// TwinCAT 3 PLC project TcoCoreTests
// Title: TcoCoreTests
// Company: Vortex.Library
// ProjectVersion: 0.6.0.913
// ProgramVersion: 3.1.4024.12
// libraries:
//   Tc2_EtherCAT, * (Beckhoff Automation GmbH)
//   Tc2_Standard, * (Beckhoff Automation GmbH)
//   Tc2_System, * (Beckhoff Automation GmbH)
//   Tc3_Module, * (Beckhoff Automation GmbH)
//   TcoCore, 0.6.0.913 (Vortex.Library)
// project tree:
//   Components/ fbPiston.TcPOU, fbPistonConfig.TcDUT, fbPistonMoveTask.TcPOU, fbPistonStatus.TcDUT, IPistonGripper.TcIO, IPistonHorizontal.TcIO, IPistonVertical.TcIO
//   / PlcTask1.TcTTO
//   POUs/ MAIN.TcPOU
//   Tests/TcoComponent/PlcExecuted/ eTcoComponentTests.TcDUT, TcoComponentTestContext.TcPOU, TestComponent.TcPOU
//   Tests/TcoComponent/ TcoComponentTest.TcPOU, _TcoComponent.TcPOU
//   Tests/TcoContext/ TcoContextTest.TcPOU
//   Tests/TcoLogger/PlcExecuted/ eTcoLoggerTests.TcDUT, TcoLoggerTestContext.TcPOU, TcoLoggerTest.TcPOU
//   Tests/TcoMessenger/ TcoContextMessagingPerf.TcPOU, TcoMessengerContextTest.TcPOU, TcoMessengerTests.TcPOU
//   Tests/TcoObject/EqualsOverride/ TcoObjectEqualsTest.TcPOU
//   Tests/TcoObject/ TcoObjectTest.TcPOU
//   Tests/TcoRemoteTask/PlcExecuted/ eTcoRemoteTaskTests.TcDUT, TcoRemoteTaskTest.TcPOU, TcoRemoteTaskTestContext.TcPOU
//   Tests/TcoRtc/ TcoRtcTest.TcPOU
//   Tests/TcoSequenceObserver/ eTcoSequenceObserverTests.TcDUT, TcoSequenceObserverTests.TcPOU
//   Tests/TcoSequencer/PlcExecuted/ eTcoSequencerTests.TcDUT, TcoSequencerTestChildState.TcPOU, TcoSequencerTestContext.TcPOU, TcoSequencerTestType.TcPOU
//   Tests/TcoSequencer/ TcoSequencerAutoRestorableTest.TcPOU, TcoSequencerNonAutoRestorableTest.TcPOU, _TcoSequencer.TcPOU
//   Tests/TcoSequence/PlcExecuted/ eTcoSequenceTests.TcDUT, TcoSequenceTestChildState.TcPOU, TcoSequenceTestContext.TcPOU, TcoSequenceTestType.TcPOU
//   Tests/TcoSequence/ TcoSequenceAutoRestorableTest.TcPOU, TcoSequenceNonAutoRestorableTest.TcPOU, _TcoSequence.TcPOU
//   Tests/TcoState/ TcoStateTest.TcPOU, TcoStateAutoRestoreTest.TcPOU
//   Tests/TcoTask/PlcExecuted/ eTcoTaskTests.TcDUT, TcoTaskPlcTestState.TcPOU, TcoTaskPlcTestObject.TcPOU, TcoTaskPlcTest.TcPOU, TcoTaskTestContext.TcPOU
//   Tests/TcoTask/ TcoTaskTest.TcPOU
//   Tests/TcoToggleTask/ eTcoToggleTaskTests.TcDUT, TcoToggleTaskTestContext.TcPOU, TcoToggleTaskTests.TcPOU
//   Tests/Utilities/ StringBuilderTests.TcPOU
// (motion and I/O tree: see PLC project tcocore)
// real-time tasks:
//   TASK PlcTask: cycle T#10ms, priority 20, ADS port 350
//   TASK PlcTask1: cycle T#10ms, priority 21, ADS port 351
//   TASK PlcTask2: cycle T#10ms, priority 22, ADS port 352

CONFIGURATION TcoCoreTests
    RESOURCE PLC ON TwinCAT3
        TASK PlcTask1(INTERVAL := T#10ms, PRIORITY := 21);
        PROGRAM MAIN WITH PlcTask1 : MAIN;
    END_RESOURCE
END_CONFIGURATION

// ---- Components/fbPistonConfig.TcDUT
TYPE fbPistonConfig :
STRUCT
    MaxTimeToReachHome : TIME;
    MaxTimeToReachWork : TIME;
END_STRUCT
END_TYPE

// ---- Components/fbPistonStatus.TcDUT
TYPE fbPistonStatus :
STRUCT
    AtHome : TIME;
    AtWork : TIME;
END_STRUCT
END_TYPE

// ---- Tests/TcoComponent/PlcExecuted/eTcoComponentTests.TcDUT
{attribute 'qualified_only'}
{attribute 'strict'}
TYPE eTcoComponentTests :
(
    GetSignalInfo := 100
);
END_TYPE

// ---- Tests/TcoLogger/PlcExecuted/eTcoLoggerTests.TcDUT
{attribute 'qualified_only'}
{attribute 'strict'}
TYPE eTcoLoggerTests :
(
    PushMessage := 10,
    PushMessageMultiple := 20,
    PushMessageMultipleInMoreCycles := 30,
    SimplePush := 40
);
END_TYPE

// ---- Tests/TcoRemoteTask/PlcExecuted/eTcoRemoteTaskTests.TcDUT
{attribute 'qualified_only'}
{attribute 'strict'}
TYPE eTcoRemoteTaskTests :
(
    RestoreTasks := 10,
    InvokeInitializedCSharpMethod := 100,
    InvokeNotInitializedCSharpMethod := 200,
    ExceptionInMethodWillResultInException := 400
);
END_TYPE

// ---- Tests/TcoSequenceObserver/eTcoSequenceObserverTests.TcDUT
{attribute 'qualified_only'}
{attribute 'strict'}
TYPE eTcoSequenceObserverTests :
(
    RestoreSequencer := 1,
    RunSequenceWithObserverTest := 10,
    RunSequenceWithoutObserverTest := 20
);
END_TYPE

// ---- Tests/TcoSequencer/PlcExecuted/eTcoSequencerTests.TcDUT
{attribute 'qualified_only'}
{attribute 'strict'}
TYPE eTcoSequencerTests :
(
    none := -1,
    CallSequencerBodiesOnly := 100,
    RestoreSequencers,
    NumberOfStepsCount := 500,
    ExecutionInOnePLCcycle := 501,
    OnStepCompleted := 502,
    OnSequenceCompleted := 503,
    RestoreChildBetweenSteps := 504,
    OnStateChangeWithRestoreCallInside := 505,
    MinStepId := 506,
    MaxStepId := 507,
    RequestStepToFirstStepWithStepId0 := 508,
    RequestStep := 509,
    CheckStepIdUniqueness := 510,
    RestoreAlreadyCheckedSequence := 512,
    NotUniqueStepId := 513,
    AfterErrorRestore := 516,
    ChangeStepIdDuringExecution := 520,
    CommentOutPartOfRunningSequencer := 524,
    UncommentPartOfRunningSequencer := 526,
    OpenCloseSequence := 530,
    RequestStepFromLowerToHigher := 541,
    RequestStepFromHigherToLower := 542,
    RequestStepToNotExistingStep := 544,
    RequestStepWhilePreviousRequestStepHasNotBeenYetProcessed := 547,
    DisableStepEnabledAndActiveInPreviousPLCcycle := 551,
    RequestStepCallingCyclically := 560,
    SetStepMode := 570,
    StepMode := 580,
    InvalidMode := 582,
    StepInError := 583,
    CheckStepIdUniquenessStepMode := 590,
    NotUniqueStepIdInStepMode := 594,
    AfterErrorResetInStepMode := 597,
    InvalidModeDetailed := 602,
    StepInErrorDetailed := 604,
    StepModeStepIn := 611,
    StepModeChangeStepIdDuringExecution := 612,
    StepModeChangeStepOrder := 615,
    StepModeCommentOutPartOfRunningSequencer := 618,
    StepModeUncommentPartOfRunningSequencer := 621,
    StepModeRequestStepFromLowerToHigher := 631,
    StepModeRequestStepFromHigherToLower := 633,
    StepModeRequestStepToNotExistingStep := 635,
    StepModeRequestStepWhilePreviousRequestStepHasnotBeenYetProcessed := 640,
    StepModeDisabledStep := 641,
    StepModeStepForwardBackward := 670,
    StepModeStepInDetailed := 681,
    SwitchStepModeOnDuringStepExecution := 691,
    StepModeStepForwardFromRunningStep := 693,
    StepModeStepBackwardFromRunningStep := 695,
    SwitchStepModeStepOffFromReadyToRun := 696,
    SwitchStepModeStepOnFromRunning := 697,
    SwitchStepModeStepOffFromRunning := 698,
    OnStateChangeWhenChangingModes := 699
);
END_TYPE

// ---- Tests/TcoSequence/PlcExecuted/eTcoSequenceTests.TcDUT
{attribute 'qualified_only'}
{attribute 'strict'}
TYPE eTcoSequenceTests :
(
    none := -1,
    Initialize := 10,
    CallSequencerBodiesOnly := 100,
    RestoreSequencers,
    NumberOfStepsCount := 500,
    ExecutionInOnePLCcycle := 501,
    OnStepCompleted := 502,
    OnSequenceCompleted := 503,
    RestoreChildBetweenSteps := 504,
    OnStateChangeWithRestoreCallInside := 505,
    MinStepId := 506,
    MaxStepId := 507,
    RequestStepToFirstStepWithStepId0 := 508,
    RequestStep := 509,
    CheckStepIdUniqueness := 510,
    RestoreAlreadyCheckedSequence := 512,
    NotUniqueStepId := 513,
    AfterErrorRestore := 516,
    ChangeStepIdDuringExecution := 520,
    CommentOutPartOfRunningSequencer := 524,
    UncommentPartOfRunningSequencer := 526,
    OpenCloseSequence := 530,
    RequestStepFromLowerToHigher := 541,
    RequestStepFromHigherToLower := 542,
    RequestStepToNotExistingStep := 544,
    RequestStepWhilePreviousRequestStepHasNotBeenYetProcessed := 547,
    DisableStepEnabledAndActiveInPreviousPLCcycle := 551,
    RequestStepCallingCyclically := 560,
    SetStepMode := 570,
    StepMode := 580,
    InvalidMode := 582,
    StepInError := 583,
    CheckStepIdUniquenessStepMode := 590,
    NotUniqueStepIdInStepMode := 594,
    AfterErrorResetInStepMode := 597,
    InvalidModeDetailed := 602,
    StepInErrorDetailed := 604,
    StepModeStepIn := 611,
    StepModeChangeStepIdDuringExecution := 612,
    StepModeChangeStepOrder := 615,
    StepModeCommentOutPartOfRunningSequencer := 618,
    StepModeUncommentPartOfRunningSequencer := 621,
    StepModeRequestStepFromLowerToHigher := 631,
    StepModeRequestStepFromHigherToLower := 633,
    StepModeRequestStepToNotExistingStep := 635,
    StepModeRequestStepWhilePreviousRequestStepHasnotBeenYetProcessed := 640,
    StepModeDisabledStep := 641,
    StepModeStepForwardBackward := 670,
    StepModeStepInDetailed := 681,
    SwitchStepModeOnDuringStepExecution := 691,
    StepModeStepForwardFromRunningStep := 693,
    StepModeStepBackwardFromRunningStep := 695,
    SwitchStepModeStepOffFromReadyToRun := 696,
    SwitchStepModeStepOnFromRunning := 697,
    SwitchStepModeStepOffFromRunning := 698,
    OnStateChangeWhenChangingModes := 699,
    MissedSequenceOpening := 6100,
    MissedSequenceClosing := 6200,
    FreshStateEntry := 6300
);
END_TYPE

// ---- Tests/TcoTask/PlcExecuted/eTcoTaskTests.TcDUT
{attribute 'qualified_only'}
{attribute 'strict'}
TYPE eTcoTaskTests :
(
    CallTasksBodiesOnly := 100,
    RestoreTasks,
    TaskInvokeAndWaitForDone := 300,
    TaskInvokeAfterDoneWithNoEmptyCycles,
    TaskInvokeAfterDoneWithOneEmptyCycle,
    TaskInvokeAfterDoneWithAbortCall,
    TaskInvokeAfterDoneWithRestoreCall,
    TaskAbortDuringExecutionAndInvoke,
    TaskError := 310,
    TaskInvokeAfterErrorNoRestoreNoEmptyCycles,
    TaskInvokeAfterErrorNoRestoreOneEmptyCycle,
    TaskInvokeAfterErrorWithRestore,
    TaskAbortDuringExecution,
    TaskMessage,
    IdentitiesTest,
    CheckAutoRestoreProperties,
    AutoRestoreOnStateChange,
    InvokeDisabledTask := 320,
    DisableExecutingTask,
    InvokeTaskThenDisable,
    DisableTaskInErrorStateEnableAndTriggerAgain,
    ElapsedTypeMeasurement := 330,
    TaskExecutingWithDoneAndErrorStatement := 340,
    TaskExecutingWithErrorAndDoneStatement := 350,
    TaskExecuteMethodNotCalled := 360,
    TaskExecuteMethodCalled := 370
);
END_TYPE

// ---- Tests/TcoToggleTask/eTcoToggleTaskTests.TcDUT
{attribute 'qualified_only'}
{attribute 'strict'}
TYPE eTcoToggleTaskTests :
(
    Reinit := 1001,
    CleanUp := 1002,
    Message := 1003,
    TriggerToggleWhileRunNotCalled := 1004,
    TriggerToggleWhileDisabled := 1005,
    TriggerToggleWhileEnabled := 1006,
    TriggerOnWhileRunNotCalled := 1007,
    TriggerOnWhileDisabled := 1008,
    TriggerOnWhileEnabled := 1009,
    TriggerOffWhileRunNotCalled := 1010,
    TriggerOffWhileDisabled := 1011,
    TriggerOffWhileEnabled := 1012
);
END_TYPE

// ---- Components/IPistonGripper.TcIO
INTERFACE IPistonGripper

METHOD Close : TcoCore.ITcoTaskStatus
END_METHOD

METHOD Open : TcoCore.ITcoTaskStatus
END_METHOD

END_INTERFACE

// ---- Components/IPistonHorizontal.TcIO
INTERFACE IPistonHorizontal

METHOD MoveLeft : TcoCore.ITcoTaskStatus
END_METHOD

METHOD MoveRight : TcoCore.ITcoTaskStatus
END_METHOD

END_INTERFACE

// ---- Components/IPistonVertical.TcIO
INTERFACE IPistonVertical

METHOD MoveDown : TcoCore.ITcoTaskStatus
END_METHOD

METHOD MoveUp : TcoCore.ITcoTaskStatus
END_METHOD

END_INTERFACE

// ---- POUs/MAIN.TcPOU
PROGRAM MAIN
VAR
    //TcRpc tests
    _tcoRtcTest_A : TcoRtcTest;
    _tcoRtcTest_B : TcoRtcTest;
    _tcoContextTest_A : TcoContextTest;
    _tcoContextTest_B : TcoContextTest;
    _tcoSequencerAutoRestorableTest : TcoSequencerAutoRestorableTest;
    _tcoSequencerNonAutoRestorableTest : TcoSequencerNonAutoRestorableTest;
    _tcoSequenceAutoRestorableTest : TcoSequenceAutoRestorableTest;
    _tcoSequenceNonAutoRestorableTest : TcoSequenceNonAutoRestorableTest;
    _tcoMessengerContextTest : TcoMessengerContextTest;
    _tcoContextMessagingPerf : TcoContextMessagingPerf;
    _tcoComponentTest : TcoComponentTest;
    _stringBuilderTest : StringBuilderTests;
    //PLC executed tests
    _tcoTaskTestContext : TcoTaskTestContext;
    _tcoToggleTaskTestContext : TcoToggleTaskTestContext;
    {attribute addProperty Name "Test base component class"}
    _tcoComponentTestContext : TcoComponentTestContext;
    _tcoRemoteTaskTestContext : TcoRemoteTaskTestContext;
    _tcoSequencerTestContext : TcoSequencerTestContext;
    _tcoSequenceTestContext : TcoSequenceTestContext;
    _tcoLoggerTestContext : TcoLoggerTestContext;
    _tcoSequenceObserverTests : TcoSequenceObserverTests;
END_VAR

//TcRpc tests
_tcoRtcTest_A();
_tcoRtcTest_B();
_tcoContextTest_A();
_tcoContextTest_B();
_tcoSequencerAutoRestorableTest();
_tcoSequencerNonAutoRestorableTest();
_tcoSequenceAutoRestorableTest();
_tcoSequenceNonAutoRestorableTest();
_tcoMessengerContextTest();
_tcoContextMessagingPerf();
_tcoComponentTest();
_stringBuilderTest();
//PLC executed tests
_tcoTaskTestContext.ProbeRun();
_tcoToggleTaskTestContext.ProbeRun();
_tcoComponentTestContext.ProbeRun();
_tcoRemoteTaskTestContext.ProbeRun();
_tcoSequencerTestContext.ProbeRun();
_tcoSequenceTestContext.ProbeRun();
_tcoLoggerTestContext.ProbeRun();
_tcoSequenceObserverTests.ProbeRun();

END_PROGRAM

// ---- Tests/TcoRtc/TcoRtcTest.TcPOU
FUNCTION_BLOCK TcoRtcTest EXTENDS TcoCore._internals_TcoContext
VAR
    _callMyPlcInstanceSync : BOOL := FALSE;
    _callMyPlcInstanceRun : BOOL := FALSE;
    _myIdentity : ULINT;
    _nowLocal : DATE_AND_TIME;
    _nowUtc : DATE_AND_TIME;
    _rtcIsValid : BOOL := FALSE;
    _rtcIsSynchronized : BOOL := FALSE;
    _rtcSynchParamsSet : TcoCore.RtcSynchParams;
    _rtcSynchParamsGet : TcoCore.RtcSynchParams;
END_VAR

IF THIS^._callMyPlcInstanceSync THEN
    THIS^.RtcSynchronize(_rtcSynchParamsSet.doSynch, _rtcSynchParamsSet.syncAmsId, _rtcSynchParamsSet.syncPeriod);
END_IF

IF THIS^._callMyPlcInstanceRun THEN
    THIS^.Run();
    _nowLocal := THIS^.RealTimeClock.NowLocal();
    _nowUtc := THIS^.RealTimeClock.NowUTC();
    _rtcIsValid := THIS^.RealTimeClock.IsValid;
    _rtcIsSynchronized := THIS^.RealTimeClock.IsSynchronized;
    _myIdentity := THIS^.Identity;
END_IF

{attribute 'TcRpcEnable'}
METHOD INTERNAL GetSynchParams
_rtcSynchParamsGet := SUPER^._GetSynchParams();
END_METHOD

METHOD PROTECTED Main
END_METHOD

{attribute 'TcRpcEnable'}
METHOD INTERNAL NowLocal
_nowLocal := THIS^.RealTimeClock.NowLocal();
END_METHOD

{attribute 'TcRpcEnable'}
METHOD INTERNAL NowUtc
_nowUtc := THIS^.RealTimeClock.NowUTC();
END_METHOD

{attribute 'TcRpcEnable'}
METHOD INTERNAL RtcIsSynchronized : BOOL
RtcIsSynchronized := THIS^.RealTimeClock.IsSynchronized;
_rtcIsSynchronized := THIS^.RealTimeClock.IsSynchronized;
END_METHOD

{attribute 'TcRpcEnable'}
METHOD INTERNAL RtcIsValid : BOOL
RtcIsValid := THIS^.RealTimeClock.IsValid;
_rtcIsValid := THIS^.RealTimeClock.IsValid;
END_METHOD

{attribute 'TcRpcEnable'}
METHOD INTERNAL TickClock : STRING
TickClock := Tc2_EtherCAT.DCTIME64_TO_STRING(THIS^.RealTimeClock.TickClock());
END_METHOD

END_FUNCTION_BLOCK

// ---- Tests/TcoContext/TcoContextTest.TcPOU
FUNCTION_BLOCK TcoContextTest EXTENDS TcoCore._internals_TcoContext
VAR
    _callMyPlcInstance : BOOL := FALSE;
    _startCycles : ULINT;
    _endCycles : ULINT;
    _mainCycles : ULINT;
    _tcoObjectTest_A : TcoObjectTest(THIS^);
    _tcoObjectTest_B : TcoObjectTest(THIS^);
    _tcoObjectTest_Misc : TcoObjectTest(THIS^);
    _myIdentity : ULINT;
    _onEntryCount : ULINT;
    _onExitCount : ULINT;
END_VAR

IF THIS^._callMyPlcInstance THEN
    THIS^.Run();
END_IF

{attribute 'TcRpcEnable'}
METHOD INTERNAL CallMainFromUnitTest
THIS^.Main();
END_METHOD

{attribute 'TcRpcEnable'}
METHOD INTERNAL CallRunFromUnitTest
THIS^.Run();
END_METHOD

{attribute 'TcRpcEnable'}
METHOD INTERNAL ContextClose
SUPER^._Close();
END_METHOD

{attribute 'TcRpcEnable'}
METHOD INTERNAL ContextOpen
SUPER^._Open();
END_METHOD

METHOD PROTECTED Main
_mainCycles := _mainCycles + 1;
_myIdentity := THIS^.Identity;
END_METHOD

(*~
    <docu>
        <summary>
            Called on entry into context. When overridden in derived class allows to execute an arbitrary logic prior to opening the context cycle.
            <remarks>
                <note type="important">
                    The method executes prior to opening the context. The context might not be properly initialized on first call.
                    Any information contained in the context at this point are from the last execution.
                </note>
            </remarks>
        </summary>
    </docu>
~*)
METHOD PROTECTED OnEntry
_onEntryCount := _onEntryCount + 1;
END_METHOD

(*~
    <docu>
        <summary>
            Called upon exit from the context. When overridden in derived class allows to execute an arbitrary logic after closing the context cycle.
        </summary>
    </docu>
~*)
METHOD PROTECTED OnExit
_onExitCount := _onExitCount + 1;
END_METHOD

{attribute 'TcRpcEnable'}
METHOD INTERNAL ReadOutCycleCounters
_startCycles := THIS^.StartCycleCount;
_endCycles := THIS^.EndCycleCount;
_myIdentity := THIS^.Identity;
END_METHOD

END_FUNCTION_BLOCK

// ---- Tests/TcoObject/TcoObjectTest.TcPOU
FUNCTION_BLOCK TcoObjectTest EXTENDS TcoCore.TcoObject
VAR
    _myIdentity : ULINT;
    _myContextIdentity : ULINT;
    _myContextStartCount : ULINT;
    _myContextEndCount : ULINT;
    _myParentIdentity : ULINT;
    _tcoTaskTest_A : TcoTaskTest(THIS^);
    _tcoTaskTest_B : TcoTaskTest(THIS^);
    _tcoStateTest_A : TcoStateTest(THIS^, eRestoreMode.AutoRestoreMembers);
    _tcoStateTest_B : TcoStateTest(THIS^, eRestoreMode.None);
    // Object equality
    _tcoObjectEqualsTestObj1 : TcoObjectEqualsTest(THIS^);
    _tcoObjectEqualsTestObj2 : TcoObjectEqualsTest(THIS^);
END_VAR

{attribute 'TcRpcEnable'}
METHOD INTERNAL CallTaskInstancies
_tcoTaskTest_A();
_tcoTaskTest_B();
END_METHOD

{attribute 'TcRpcEnable'}
METHOD PUBLIC EqualsOverrideTest : BOOL
EqualsOverrideTest := _tcoObjectEqualsTestObj1.EqualsTo(_tcoObjectEqualsTestObj2);
END_METHOD

{attribute 'TcRpcEnable'}
METHOD PUBLIC EqualsTest : BOOL
VAR_INPUT
    _case : INT;
END_VAR
VAR
    referenceTo_a_TcoStateTest : REFERENCE TO TcoStateTest;
END_VAR
CASE _case OF
    0:
        referenceTo_a_TcoStateTest REF= _tcoStateTest_A;
        EqualsTest := _tcoStateTest_A.EqualsTo(referenceTo_a_TcoStateTest);
    1:
        EqualsTest := _tcoStateTest_A.EqualsTo(_tcoStateTest_B);
    4:
        EqualsTest := _tcoStateTest_B.EqualsTo(_tcoStateTest_A);
    2:
        EqualsTest := _tcoObjectEqualsTestObj1.EqualsTo(_tcoObjectEqualsTestObj1);
    3:
        EqualsTest := _tcoObjectEqualsTestObj1.EqualsTo(_tcoObjectEqualsTestObj2);
END_CASE
END_METHOD

{attribute 'TcRpcEnable'}
METHOD INTERNAL ReadOutIdentities
_myIdentity := THIS^.Identity;
_myContextIdentity := THIS^.Context.Identity;
_myContextStartCount := THIS^.Context.StartCycleCount;
_myContextEndCount := THIS^.Context.EndCycleCount;
_myParentIdentity := THIS^.Parent.Identity;
END_METHOD

END_FUNCTION_BLOCK

// ---- Tests/TcoTask/TcoTaskTest.TcPOU
FUNCTION_BLOCK TcoTaskTest EXTENDS TcoCore.TcoTask
VAR
    _isBusy : BOOL;
    _isError : BOOL;
    _isDone : BOOL;
    _isReady : BOOL;
    _isInvokeRequestTrue : BOOL;
    _counterSetValue : ULINT;
    _counterValue : ULINT;
    _invokeCounter : ULINT;
    _executeCounter : ULINT;
    _doneCounter : ULINT;
    _invokeRisingEdgeCounter : ULINT;
    _executeRisingEdgeCounter : ULINT;
    _doneRisingEdgeCounter : ULINT;
    _previousState : eTaskState;
    _counterValuePV : ULINT;
    _myIdentity : ULINT;
    _myContextIdentity : ULINT;
    _myContextStartCount : ULINT;
    _myContextEndCount : ULINT;
    _myParentIdentity : ULINT;
    _autoRestoreByMyParentEnabled : BOOL;
    _onErrorCounter : ULINT;
    _whileErrorCounter : ULINT;
    _onStartCounter : ULINT;
END_VAR

ExecutionBody();

{attribute 'TcRpcEnable'}
METHOD INTERNAL Disable
THIS^.Enabled := FALSE;
END_METHOD

{attribute 'TcRpcEnable'}
METHOD INTERNAL Enable
THIS^.Enabled := TRUE;
END_METHOD

{attribute 'TcRpcEnable'}
METHOD INTERNAL ExecutionBody
IF (THIS^._taskState = eTaskState.Requested) THEN
    _invokeCounter := _invokeCounter + 1;
END_IF;

IF (THIS^._taskState = eTaskState.Requested AND _PreviousState <> eTaskState.Requested) THEN
    _counterValue := _counterSetValue;
    _counterValuePV := _counterValue;
    _invokeRisingEdgeCounter := _invokeRisingEdgeCounter + 1;
END_IF

IF (THIS^._taskState = eTaskState.Busy AND _previousState <> eTaskState.Busy) THEN
    _executeRisingEdgeCounter := _executeRisingEdgeCounter + 1;
END_IF

_previousState := THIS^._taskState;

IF (Execute()) THEN
    _executeCounter := _executeCounter + 1;
    _counterValue := _counterValue - 1;
    DoneWhen(_counterValue <= 0);
    ThrowWhen(ABS(_counterValuePV - _counterValue) > 1);
    _CounterValuePV := _counterValue;
END_IF

IF (THIS^._taskState = eTaskState.Done) THEN
    _doneCounter := _doneCounter + 1;
END_IF;

IF (THIS^._taskState = eTaskState.Done AND _previousState <> eTaskState.Done) THEN
    _doneRisingEdgeCounter := _doneRisingEdgeCounter + 1;
END_IF
END_METHOD

{attribute 'TcRpcEnable'}
METHOD INTERNAL GetMessage : STRING
GetMessage := SUPER^._messenger._mime.Text;
END_METHOD

METHOD PROTECTED OnError
_onErrorCounter := _onErrorCounter + 1;
END_METHOD

METHOD PROTECTED OnStart
_onStartCounter := _onStartCounter + 1;
END_METHOD

{attribute 'TcRpcEnable'}
METHOD INTERNAL PostMessage
VAR_INPUT
    Message : STRING;
END_VAR
THIS^.Messenger.Post(Message, eMessageCategory.Error);
END_METHOD

{attribute 'TcRpcEnable'}
METHOD INTERNAL ReadOutAutoRestoreProperties
_autoRestoreByMyParentEnabled := THIS^.AutoRestorable;
END_METHOD

{attribute 'TcRpcEnable'}
METHOD INTERNAL ReadOutIdentities
_myIdentity := THIS^.Identity;
_myContextIdentity := THIS^.Context.Identity;
_myContextStartCount := THIS^.Context.StartCycleCount;
_myContextEndCount := THIS^.Context.EndCycleCount;
_myParentIdentity := THIS^.Parent.Identity;
END_METHOD

{attribute 'TcRpcEnable'}
METHOD INTERNAL ReadOutState
_isBusy := THIS^.Busy;
_isError := THIS^.Error;
_isDone := THIS^.Done;
_isReady := THIS^.Ready;
_isInvokeRequestTrue := THIS^._invokeRequest;
END_METHOD

{attribute 'TcRpcEnable'}
METHOD INTERNAL SetInvokeRequest
THIS^._invokeRequest := TRUE;
END_METHOD

{attribute 'TcRpcEnable'}
METHOD INTERNAL SetPreviousStateToReady
THIS^._previousState := eTaskState.Ready;
END_METHOD

{attribute 'TcRpcEnable'}
METHOD INTERNAL TriggerAbort
THIS^.Abort();
END_METHOD

{attribute 'TcRpcEnable'}
METHOD INTERNAL TriggerInvoke
THIS^.Invoke();
END_METHOD

{attribute 'TcRpcEnable'}
METHOD INTERNAL TriggerRestore
THIS^.Restore();
END_METHOD

(*~
    <docu>
        <summary>
            Executes until task is in ```Error``` state .
        </summary>
    </docu>
~*)
METHOD PROTECTED WhileError
_whileErrorCounter := _whileErrorCounter + 1;
END_METHOD

END_FUNCTION_BLOCK

// ---- Tests/TcoState/TcoStateTest.TcPOU
FUNCTION_BLOCK TcoStateTest EXTENDS TcoState
VAR
    _myIdentity : ULINT;
    _myContextIdentity : ULINT;
    _myContextStartCount : ULINT;
    _myContextEndCount : ULINT;
    _myParentIdentity : ULINT;
    _myState : INT;
    _tcoTaskTest_A : TcoTaskTest(THIS^);
    _tcoTaskTest_B : TcoTaskTest(THIS^);
    _tcoStateTest_A : TcoStateAutoRestoreTest(THIS^, eRestoreMode.None);
    _tcoStateTest_B : TcoStateAutoRestoreTest(THIS^, eRestoreMode.None);
    _onStateChangeCounter : INT;
    _autoRestoreToMyChildsEnabled : BOOL;
    _autoRestoreByMyParentEnabled : BOOL;
END_VAR

{attribute 'TcRpcEnable'}
METHOD INTERNAL CallTaskInstancies
_tcoTaskTest_A();
_tcoTaskTest_B();
END_METHOD

{attribute 'TcRpcEnable'}
METHOD INTERNAL CleanUp
THIS^.ChangeState(0);
_myState := State;
_onStateChangeCounter := 0;
_autoRestoreToMyChildsEnabled := FALSE;
_autoRestoreByMyParentEnabled := FALSE;
END_METHOD

{attribute 'TcRpcEnable'}
METHOD INTERNAL GetMessage : STRING
GetMessage := SUPER^._messenger._mime.Text;
END_METHOD

METHOD PROTECTED OnStateChange
VAR_INPUT
    PreviousState : INT;
    NewState : INT;
END_VAR
VAR
    message : STRING;
END_VAR
_onStateChangeCounter := _onStateChangeCounter + 1;
message := CONCAT('My state has been change from ', INT_TO_STRING(PreviousState));
message := CONCAT(message, ' to the new state ');
message := CONCAT(message, INT_TO_STRING(NewState));
message := CONCAT(message, '.');
THIS^.Messenger.Post(message, eMessageCategory.Debug);
SUPER^.OnStateChange(PreviousState, NewState);
END_METHOD

{attribute 'TcRpcEnable'}
METHOD INTERNAL PostMessage
VAR_INPUT
    Message : STRING;
END_VAR
THIS^.Messenger.Post(Message, eMessageCategory.Debug);
END_METHOD

{attribute 'TcRpcEnable'}
METHOD INTERNAL ReadOutAutoRestoreProperties
_autoRestoreToMyChildsEnabled := THIS^.IsAutoRestoreEnabled;
_autoRestoreByMyParentEnabled := THIS^.AutoRestorable;
END_METHOD

{attribute 'TcRpcEnable'}
METHOD INTERNAL ReadOutIdentities
_myIdentity := THIS^.Identity;
_myContextIdentity := THIS^.Context.Identity;
_myParentIdentity := THIS^.Parent.Identity;
_myContextStartCount := THIS^.Context.StartCycleCount;
_myContextEndCount := THIS^.Context.EndCycleCount;
END_METHOD

{attribute 'TcRpcEnable'}
METHOD INTERNAL ReadOutState
_myState := THIS^.State;
THIS^._tcoTaskTest_A.ReadOutState();
THIS^._tcoTaskTest_B.ReadOutState();
END_METHOD

{attribute 'TcRpcEnable'}
METHOD INTERNAL TriggerChangeState
VAR_INPUT
    NewState : INT;
END_VAR
THIS^.ChangeState(NewState);
END_METHOD

{attribute 'TcRpcEnable'}
METHOD INTERNAL TriggerChangeStateWithObjectRestore
VAR_INPUT
    NewState : INT;
END_VAR
THIS^.ChangeState(NewState).RestoreObject(THIS^._tcoTaskTest_A).RestoreObject(THIS^._tcoTaskTest_B);
END_METHOD

{attribute 'TcRpcEnable'}
METHOD INTERNAL TriggerRestore
THIS^.Restore();
END_METHOD

{attribute 'TcRpcEnable'}
METHOD INTERNAL TriggerTaskInvoke
THIS^._tcoTaskTest_A.Invoke();
THIS^._tcoTaskTest_B.Invoke();
END_METHOD

END_FUNCTION_BLOCK

// ---- Tests/TcoState/TcoStateAutoRestoreTest.TcPOU
FUNCTION_BLOCK TcoStateAutoRestoreTest EXTENDS TcoState
VAR
    _myState : INT;
    _onStateChangeCounter : INT;
    _restoreCounter : INT;
    _autoRestoreToMyChildsEnabled : BOOL;
    _autoRestoreByMyParentEnabled : BOOL;
    _countsPerStep : ULINT;
    _counterValue : ULINT;
END_VAR

{attribute 'TcRpcEnable'}
METHOD INTERNAL CleanUp
THIS^.ChangeState(0);
_myState := State;
_onStateChangeCounter := 0;
_restoreCounter := 0;
_autoRestoreToMyChildsEnabled := FALSE;
_autoRestoreByMyParentEnabled := FALSE;
_countsPerStep := 0;
_counterValue := 0;
END_METHOD

{attribute 'TcRpcEnable'}
METHOD INTERNAL ExecutionBody
IF State = -1 THEN
    _counterValue := 0;
    ChangeState(0);
END_IF

IF State = 0 THEN
    _counterValue := _counterValue + 1;

    IF (_counterValue MOD _countsPerStep) = 0 THEN
        ChangeState(State + 10);
    END_IF
END_IF

IF State = 10 THEN
    _counterValue := _counterValue + 1;

    IF (_counterValue MOD _countsPerStep) = 0 THEN
        ChangeState(State + 10);
    END_IF
END_IF

IF State = 20 THEN
    _counterValue := _counterValue + 1;

    IF (_counterValue MOD _countsPerStep) = 0 THEN
        ChangeState(State + 10);
    END_IF
END_IF

IF State = 30 THEN
    _counterValue := _counterValue + 1;

    IF (_counterValue MOD _countsPerStep) = 0 THEN
        ChangeState(State + 10);
    END_IF
END_IF

IF State = 40 THEN
    _counterValue := _counterValue + 1;

    IF (_counterValue MOD _countsPerStep) = 0 THEN
        ChangeState(State + 10);
    END_IF
END_IF

IF State = 50 THEN
    _counterValue := _counterValue + 1;

    IF (_counterValue MOD _countsPerStep) = 0 THEN
        ChangeState(State + 10);
    END_IF
END_IF

IF State = 60 THEN
    ChangeState(-1);
END_IF

_myState := State;
END_METHOD

METHOD PROTECTED OnStateChange
VAR_INPUT
    PreviousState : INT;
    NewState : INT;
END_VAR
_onStateChangeCounter := _onStateChangeCounter + 1;
SUPER^.OnStateChange(PreviousState, NewState);
END_METHOD

{attribute 'TcRpcEnable'}
METHOD INTERNAL ReadOutAutoRestoreProperties
_autoRestoreToMyChildsEnabled := THIS^.IsAutoRestoreEnabled;
_autoRestoreByMyParentEnabled := THIS^.AutoRestorable;
END_METHOD

METHOD Restore : ITcoRestorable
_restoreCounter := _restoreCounter + 1;
SUPER^.Restore();
END_METHOD

{attribute 'TcRpcEnable'}
METHOD INTERNAL TriggerRestore
THIS^.Restore();
_myState := State;
END_METHOD

END_FUNCTION_BLOCK

// ---- Tests/TcoObject/EqualsOverride/TcoObjectEqualsTest.TcPOU
FUNCTION_BLOCK TcoObjectEqualsTest EXTENDS TcoCore.TcoObject
VAR
    _someNumber : INT;
    _someString : STRING;
END_VAR

METHOD PUBLIC EqualsTo : BOOL
VAR_INPUT
    Object : ITcoObject;
END_VAR
VAR
    _object : POINTER TO TcoObjectEqualsTest;
END_VAR
IF (__QUERYPOINTER(Object, _object)) THEN
    EqualsTo := _object^._someNumber = THIS^._someNumber AND _object^._someString = THIS^._someString;
END_IF;
END_METHOD

PROPERTY SomeNumber : INT
GET
SomeNumber := _someNumber;
END_GET
SET
_someNumber := SomeNumber;
END_SET
END_PROPERTY

PROPERTY SomeString : STRING
GET
SomeString := _someString;
END_GET
SET
_someString := SomeString;
END_SET
END_PROPERTY

END_FUNCTION_BLOCK

// ---- Tests/TcoSequencer/TcoSequencerAutoRestorableTest.TcPOU
FUNCTION_BLOCK TcoSequencerAutoRestorableTest EXTENDS TcoCore._internals_TcoContext
VAR
    _callMyPlcInstance : BOOL := FALSE;
    _sequencer : _TcoSequencer(THIS^, eRestoreMode.AutoRestoreMembers);
    _runPLCinstanceOnce : BOOL := FALSE;
    _runPLCinstanceCyclicaly : BOOL := FALSE;
    _stepID : INT := 32764;
    _enabled : BOOL;
    _stepDescription : STRING := 'Last step sequence message';
    _runOneStep : BOOL;
    _runAllSteps : BOOL;
    _finishStep : BOOL;
    _restore : BOOL;
    _cycleCount : INT;
    _restoreCycleCount : INT;
    _init : BOOL;
    _setCurrentStepPropTestData : TcoCore.StepDetails;
END_VAR

IF _callMyPlcInstance THEN
    IF NOT _init THEN
        ContextOpen();
        ContextClose();
        _init := THIS^._rtc.IsValid;
    END_IF

    IF _restore THEN
        ContextOpen();
        THIS^._sequencer.Restore();
        _restoreCycleCount := _restoreCycleCount + 1;
        _restore := FALSE;
        ContextClose();
        RETURN;
    END_IF

    IF _runPLCinstanceOnce AND NOT _runPLCinstanceCyclicaly THEN
        ContextOpen();
        THIS^.PLCinstanceRun(_stepID, _enabled, _stepDescription);
        _cycleCount := _cycleCount + 1;
        _runPLCinstanceOnce := FALSE;
        ContextClose();
    END_IF

    IF _runPLCinstanceCyclicaly AND NOT _runPLCinstanceOnce THEN
        ContextOpen();
        THIS^.PLCinstanceRun(_stepID, _enabled, _stepDescription);
        _cycleCount := _cycleCount + 1;
        ContextClose();
    END_IF
END_IF;

{attribute 'TcRpcEnable'}
METHOD ChildHasAutoRestoreEnabled : BOOL;
ChildHasAutoRestoreEnabled := _sequencer.ChildHasAutoRestoreEnabled();
END_METHOD

{attribute 'TcRpcEnable'}
METHOD ChildIsAutoRestorable : BOOL;
ChildIsAutoRestorable := _sequencer.ChildIsAutoRestorable();
END_METHOD

{attribute 'TcRpcEnable'}
METHOD CleanupPointers
_sequencer.CleanupPointers();
END_METHOD

{attribute 'TcRpcEnable'}
METHOD ClearNumberOfSteps
_sequencer.ClearNumberOfSteps();
END_METHOD

{attribute 'TcRpcEnable'}
METHOD PROTECTED ContextClose
SUPER^._Close();
END_METHOD

{attribute 'TcRpcEnable'}
METHOD ContextOpen
SUPER^._Open();
END_METHOD

{attribute 'TcRpcEnable'}
METHOD GetChildState : INT
GetChildState := _sequencer.GetChildState();
END_METHOD

{attribute 'TcRpcEnable'}
METHOD GetCurrentStepOrder : UINT
GetCurrentStepOrder := _sequencer._currentStep.Order;
END_METHOD

{attribute 'TcRpcEnable'}
METHOD GetCurrentStepPropTest
_setCurrentStepPropTestData := THIS^._sequencer.CurrentStep;
END_METHOD

{attribute 'TcRpcEnable'}
METHOD GetNumberOfStepsInSequence : UINT
GetNumberOfStepsInSequence := _sequencer._numberOfStepsInSequence;
END_METHOD

{attribute 'TcRpcEnable'}
METHOD GetOrderOfTheCurrentlyEvaluatedStep : UINT
GetOrderOfTheCurrentlyEvaluatedStep := _sequencer._theOrderOfTheCurrentlyEvaluatedStep;
END_METHOD

{attribute 'TcRpcEnable'}
METHOD GetOrderOfTheCurrentlyExecutedStep : UINT
GetOrderOfTheCurrentlyExecutedStep := _sequencer._theOrderOfTheCurrentlyExecutedStep;
END_METHOD

{attribute 'TcRpcEnable'}
METHOD GetPreviousNumberOfStepsInSequence : UINT
GetPreviousNumberOfStepsInSequence := _sequencer._previousNumberOfStepsInSequence;
END_METHOD

{attribute 'TcRpcEnable'}
METHOD GetRequestStepCycle : UINT
GetRequestStepCycle := _sequencer.RequestStepCycle;
END_METHOD

{attribute 'TcRpcEnable'}
METHOD GetSequencerErrorId : INT
GetSequencerErrorId := _sequencer.GetSequencerErrorId();
END_METHOD

{attribute 'TcRpcEnable'}
METHOD GetTextOfTheMostImportantMessage : STRING(254)
GetTextOfTheMostImportantMessage := THIS^._sequencer.GetTextOfTheMostImportantMessage();
END_METHOD

{attribute 'TcRpcEnable'}
METHOD HasAutoRestoreEnabled : BOOL;
HasAutoRestoreEnabled := _sequencer.HasAutoRestoreEnabled();
END_METHOD

{attribute 'TcRpcEnable'}
METHOD IsAutoRestorable : BOOL;
IsAutoRestorable := _sequencer.IsAutoRestorable();
END_METHOD

{attribute 'TcRpcEnable'}
METHOD IsFirstStepEntry : BOOL
IsFirstStepEntry := THIS^._sequencer.IsFirstStepEntry();
END_METHOD

METHOD PROTECTED Main
END_METHOD

{attribute 'TcRpcEnable'}
METHOD PLCinstanceRun
VAR_INPUT
    inStepId : UINT;
    inEnabled : BOOL;
    inStepDescription : STRING(254);
END_VAR
THIS^._sequencer.SetTestParams(_runOneStep,
    _runAllSteps,
    _finishStep,
    inStepId,
    inEnabled,
    inStepDescription);

THIS^._sequencer.Run();
END_METHOD

{attribute 'TcRpcEnable'}
METHOD RequestStep
VAR_INPUT
    inRequestedStepId : INT;
END_VAR
_sequencer._RequestStep(inRequestedStepId);
END_METHOD

{attribute 'TcRpcEnable'}
METHOD Restore
_sequencer.Restore();
END_METHOD

{attribute 'TcRpcEnable'}
METHOD SequenceComplete
_sequencer._SequenceComplete();
END_METHOD

{attribute 'TcRpcEnable'}
METHOD SequencerClose
THIS^._sequencer.SequencerClose();
END_METHOD

{attribute 'TcRpcEnable'}
METHOD SequencerHasError : BOOL
SequencerHasError := _sequencer.SequencerHasError();
END_METHOD

{attribute 'TcRpcEnable'}
METHOD SequencerOpen
THIS^._sequencer.SequencerOpen();
END_METHOD

{attribute 'TcRpcEnable'}
METHOD SetChildState
VAR_INPUT
    inState : INT;
END_VAR
_sequencer.SetChildState(inState);
END_METHOD

{attribute 'TcRpcEnable'}
METHOD SetCurrentStep
VAR_INPUT
    inStepID : INT;
    inStepDescription : STRING(254);
END_VAR
_sequencer.SetCurrentStep(inStepID := inStepID, inStepDescription := inStepDescription);
END_METHOD

{attribute 'TcRpcEnable'}
METHOD SetCurrentStepToErrorState : BOOL
SetCurrentStepToErrorState := _sequencer.SetCurrentStepToErrorState();
END_METHOD

{attribute 'TcRpcEnable'}
METHOD SetCyclicMode : BOOL
SetCyclicMode := _sequencer.SetCyclicMode();
END_METHOD

{attribute 'TcRpcEnable'}
METHOD SetInvalidMode : BOOL
SetInvalidMode := _sequencer.SetInvalidMode();
END_METHOD

{attribute 'TcRpcEnable'}
METHOD SetNumberOfSteps : UINT
VAR_INPUT
    inNumberOfSteps : UINT;
END_VAR
_sequencer.SetNumberOfSteps(inNumberOfSteps);
SetNumberOfSteps := _sequencer._numberOfStepsInSequence;
END_METHOD

{attribute 'TcRpcEnable'}
METHOD SetRequestStepCycle : UINT
VAR_INPUT
    Value : UINT;
END_VAR
_sequencer.RequestStepCycle := Value;
SetRequestStepCycle := _sequencer.RequestStepCycle;
END_METHOD

{attribute 'TcRpcEnable'}
METHOD SetSequenceAsChecked : BOOL
VAR_INPUT
END_VAR
_sequencer.SetSequenceAsChecked();
END_METHOD

{attribute 'TcRpcEnable'}
METHOD SetSequenceAsNotChecked : BOOL
VAR_INPUT
END_VAR
_sequencer.SetSequenceAsNotChecked();
END_METHOD

{attribute 'TcRpcEnable'}
METHOD SetStepMode : BOOL
SetStepMode := _sequencer.SetStepMode();
END_METHOD

{attribute 'TcRpcEnable'}
METHOD Step : BOOL
VAR_INPUT
    inStepId : INT;
    inEnabled : BOOL;
    inStepDescription : STRING(254);
END_VAR
Step := _sequencer._Step(inStepID := inStepId, inEnabled := inEnabled, inStepDescription := inStepDescription);
END_METHOD

{attribute 'TcRpcEnable'}
METHOD StepBackward
_sequencer._StepBackward();
END_METHOD

{attribute 'TcRpcEnable'}
METHOD StepCompleteWhen
VAR_INPUT
    inCondition : BOOL;
END_VAR
_sequencer._StepCompleteWhen(inCondition);
END_METHOD

{attribute 'TcRpcEnable'}
METHOD StepForward
_sequencer._StepForward();
END_METHOD

{attribute 'TcRpcEnable'}
METHOD StepIn
_sequencer._StepIn();
END_METHOD

{attribute 'TcRpcEnable'}
METHOD UpdateCurrentStepDetails
VAR_INPUT
END_VAR
_sequencer.UpdateCurrentStepDetails();
END_METHOD

END_FUNCTION_BLOCK

// ---- Tests/TcoSequencer/_TcoSequencer.TcPOU
FUNCTION_BLOCK _TcoSequencer EXTENDS TcoCore._internals_TcoSequencer
VAR
    _runOneStep : BOOL;
    _runAllSteps : BOOL;
    _finishStep : BOOL;
    _stepId : INT;
    _enabled : BOOL;
    _stepDescription : STRING(254);
    _currentStepId : INT;
    _currentStepOrder : UINT;
    _currentStepEnabled : BOOL;
    _currentStepDescription : STRING(254);
    _currentStepStatus : INT;
    _currentStepDuration : TIME;
    _myTcoState : TcoState(THIS^, eRestoreMode.None);
    _onCompleteStepCount : INT;
    _onSequenceCompleteCount : INT;
    _onSequencerErrorCount : ULINT;
    _onStateChangeCount : ULINT;
    _stateChangeFrom : INT;
    _stateChangeTo : INT;
    _callRestoreInOnStateChange : BOOL;
END_VAR

METHOD _RequestStep
VAR_INPUT
    inRequestedStepId : INT;
END_VAR
THIS^.RequestStep(inRequestedStepId);
END_METHOD

METHOD _SequenceComplete
THIS^.CompleteSequence();
END_METHOD

METHOD INTERNAL _Step : BOOL
VAR_INPUT
    inStepId : INT;
    inEnabled : BOOL;
    inStepDescription : STRING(254);
END_VAR
_Step := SUPER^.Step(inStepID := inStepId, inEnabled := inEnabled, inStepDescription := inStepDescription);
END_METHOD

METHOD _StepBackward
THIS^.ModeController.StepBackward();
END_METHOD

METHOD _StepCompleteWhen
VAR_INPUT
    inCondition : BOOL;
END_VAR
THIS^.StepCompleteWhen(inCondition);
END_METHOD

METHOD _StepForward
THIS^.ModeController.StepForward();
END_METHOD

METHOD INTERNAL _StepIn
THIS^.ModeController.StepIn();
END_METHOD

METHOD INTERNAL ChildHasAutoRestoreEnabled : BOOL
ChildHasAutoRestoreEnabled := THIS^._myTcoState.IsAutoRestoreEnabled;
END_METHOD

METHOD INTERNAL ChildIsAutoRestorable : BOOL
ChildIsAutoRestorable := THIS^._myTcoState.AutoRestorable;
END_METHOD

METHOD INTERNAL CleanupPointers
IF (_pPreviusSteps <> 0) THEN
    __DELETE(_pPreviusSteps);
END_IF
END_METHOD

METHOD INTERNAL ClearNumberOfSteps
_stepCounter := 0;
_numberOfStepsInSequence := 0;
_previousNumberOfStepsInSequence := 0;
END_METHOD

METHOD INTERNAL GetChildState : INT
GetChildState := THIS^._myTcoState.State;
END_METHOD

{attribute 'TcRpcEnable'}
METHOD GetNumberOfStepsInSequence : UINT
GetNumberOfStepsInSequence := THIS^._numberOfStepsInSequence;
END_METHOD

METHOD INTERNAL GetSequencerErrorId : INT
GetSequencerErrorId := SUPER^._sequencerErrorId;
END_METHOD

METHOD INTERNAL GetTextOfTheMostImportantMessage : STRING(254)
GetTextOfTheMostImportantMessage := THIS^._messenger._mime.Text;
END_METHOD

METHOD INTERNAL HasAutoRestoreEnabled : BOOL
HasAutoRestoreEnabled := SUPER^.IsAutoRestoreEnabled;
END_METHOD

METHOD INTERNAL IsAutoRestorable : BOOL
IsAutoRestorable := SUPER^.AutoRestorable;
END_METHOD

METHOD INTERNAL IsFirstStepEntry : BOOL
IsFirstStepEntry := _isFirstStepEntry;
END_METHOD

METHOD PROTECTED Main : BOOL
//******************************************************************
IF SUPER^.Step(0, TRUE, 'Step number 0') THEN
    SUPER^.StepCompleteWhen((_runOneStep OR _runAllSteps) AND _finishStep);

    IF _runOneStep THEN
        _runOneStep := FALSE;
        RETURN;
    END_IF
END_IF

IF SUPER^.Step(1, TRUE, 'Step number 1') THEN
    SUPER^.StepCompleteWhen((_runOneStep OR _runAllSteps) AND _finishStep);

    IF _runOneStep THEN
        _runOneStep := FALSE;
        RETURN;
    END_IF
END_IF

IF SUPER^.Step(2, TRUE, 'Step number 2') THEN
    SUPER^.StepCompleteWhen((_runOneStep OR _runAllSteps) AND _finishStep);

    IF _runOneStep THEN
        _runOneStep := FALSE;
        RETURN;
    END_IF
END_IF

IF SUPER^.Step(3, TRUE, 'Step number 3') THEN
    SUPER^.StepCompleteWhen((_runOneStep OR _runAllSteps) AND _finishStep);

    IF _runOneStep THEN
        _runOneStep := FALSE;
        RETURN;
    END_IF
END_IF

IF SUPER^.Step(4, TRUE, 'Step number 4') THEN
    SUPER^.StepCompleteWhen((_runOneStep OR _runAllSteps) AND _finishStep);

    IF _runOneStep THEN
        _runOneStep := FALSE;
        RETURN;
    END_IF
END_IF

IF SUPER^.Step(5, TRUE, 'Step number 5') THEN
    SUPER^.StepCompleteWhen((_runOneStep OR _runAllSteps) AND _finishStep);

    IF _runOneStep THEN
        _runOneStep := FALSE;
        RETURN;
    END_IF
END_IF

IF SUPER^.Step(6, TRUE, 'Step number 6') THEN
    SUPER^.StepCompleteWhen((_runOneStep OR _runAllSteps) AND _finishStep);

    IF _runOneStep THEN
        _runOneStep := FALSE;
        RETURN;
    END_IF
END_IF

IF SUPER^.Step(7, TRUE, 'Step number 7') THEN
    SUPER^.StepCompleteWhen((_runOneStep OR _runAllSteps) AND _finishStep);

    IF _runOneStep THEN
        _runOneStep := FALSE;
        RETURN;
    END_IF
END_IF

IF SUPER^.Step(8, TRUE, 'Step number 8') THEN
    SUPER^.StepCompleteWhen((_runOneStep OR _runAllSteps) AND _finishStep);

    IF _runOneStep THEN
        _runOneStep := FALSE;
        RETURN;
    END_IF
END_IF

IF SUPER^.Step(9, TRUE, 'Step number 9') THEN
    SUPER^.StepCompleteWhen((_runOneStep OR _runAllSteps) AND _finishStep);

    IF _runOneStep THEN
        _runOneStep := FALSE;
        RETURN;
    END_IF
END_IF

IF SUPER^.Step(10, TRUE, 'Step number 10') THEN
    SUPER^.StepCompleteWhen((_runOneStep OR _runAllSteps) AND _finishStep);

    IF _runOneStep THEN
        _runOneStep := FALSE;
        RETURN;
    END_IF
END_IF

IF SUPER^.Step(11, TRUE, 'Step number 11') THEN
    SUPER^.StepCompleteWhen((_runOneStep OR _runAllSteps) AND _finishStep);

    IF _runOneStep THEN
        _runOneStep := FALSE;
        RETURN;
    END_IF
END_IF

IF SUPER^.Step(12, TRUE, 'Step number 12') THEN
    SUPER^.StepCompleteWhen((_runOneStep OR _runAllSteps) AND _finishStep);

    IF _runOneStep THEN
        _runOneStep := FALSE;
        RETURN;
    END_IF
END_IF

IF SUPER^.Step(13, TRUE, 'Step number 13') THEN
    SUPER^.StepCompleteWhen((_runOneStep OR _runAllSteps) AND _finishStep);

    IF _runOneStep THEN
        _runOneStep := FALSE;
        RETURN;
    END_IF
END_IF

IF SUPER^.Step(14, TRUE, 'Step number 14') THEN
    SUPER^.StepCompleteWhen((_runOneStep OR _runAllSteps) AND _finishStep);

    IF _runOneStep THEN
        _runOneStep := FALSE;
        RETURN;
    END_IF
END_IF

IF SUPER^.Step(15, TRUE, 'Step number 15') THEN
    SUPER^.StepCompleteWhen((_runOneStep OR _runAllSteps) AND _finishStep);

    IF _runOneStep THEN
        _runOneStep := FALSE;
        RETURN;
    END_IF
END_IF

IF SUPER^.Step(16, TRUE, 'Step number 16') THEN
    SUPER^.StepCompleteWhen((_runOneStep OR _runAllSteps) AND _finishStep);

    IF _runOneStep THEN
        _runOneStep := FALSE;
        RETURN;
    END_IF
END_IF

IF SUPER^.Step(17, TRUE, 'Step number 17') THEN
    SUPER^.StepCompleteWhen((_runOneStep OR _runAllSteps) AND _finishStep);

    IF _runOneStep THEN
        _runOneStep := FALSE;
        RETURN;
    END_IF
END_IF

IF SUPER^.Step(18, TRUE, 'Step number 18') THEN
    SUPER^.StepCompleteWhen((_runOneStep OR _runAllSteps) AND _finishStep);

    IF _runOneStep THEN
        _runOneStep := FALSE;
        RETURN;
    END_IF
END_IF

IF SUPER^.Step(19, TRUE, 'Step number 19') THEN
    SUPER^.StepCompleteWhen((_runOneStep OR _runAllSteps) AND _finishStep);

    IF _runOneStep THEN
        _runOneStep := FALSE;
        RETURN;
    END_IF
END_IF

IF SUPER^.Step(20, TRUE, 'Step number 20') THEN
    SUPER^.StepCompleteWhen((_runOneStep OR _runAllSteps) AND _finishStep);

    IF _runOneStep THEN
        _runOneStep := FALSE;
        RETURN;
    END_IF
END_IF

IF SUPER^.Step(21, TRUE, 'Step number 21') THEN
    SUPER^.StepCompleteWhen((_runOneStep OR _runAllSteps) AND _finishStep);

    IF _runOneStep THEN
        _runOneStep := FALSE;
        RETURN;
    END_IF
END_IF

IF SUPER^.Step(22, TRUE, 'Step number 22') THEN
    SUPER^.StepCompleteWhen((_runOneStep OR _runAllSteps) AND _finishStep);

    IF _runOneStep THEN
        _runOneStep := FALSE;
        RETURN;
    END_IF
END_IF

IF SUPER^.Step(23, TRUE, 'Step number 23') THEN
    SUPER^.StepCompleteWhen((_runOneStep OR _runAllSteps) AND _finishStep);

    IF _runOneStep THEN
        _runOneStep := FALSE;
        RETURN;
    END_IF
END_IF

IF SUPER^.Step(24, TRUE, 'Step number 24') THEN
    SUPER^.StepCompleteWhen((_runOneStep OR _runAllSteps) AND _finishStep);

    IF _runOneStep THEN
        _runOneStep := FALSE;
        RETURN;
    END_IF
END_IF

IF SUPER^.Step(25, TRUE, 'Step number 25') THEN
    SUPER^.StepCompleteWhen((_runOneStep OR _runAllSteps) AND _finishStep);

    IF _runOneStep THEN
        _runOneStep := FALSE;
        RETURN;
    END_IF
END_IF

IF SUPER^.Step(26, TRUE, 'Step number 26') THEN
    SUPER^.StepCompleteWhen((_runOneStep OR _runAllSteps) AND _finishStep);

    IF _runOneStep THEN
        _runOneStep := FALSE;
        RETURN;
    END_IF
END_IF

IF SUPER^.Step(27, TRUE, 'Step number 27') THEN
    SUPER^.StepCompleteWhen((_runOneStep OR _runAllSteps) AND _finishStep);

    IF _runOneStep THEN
        _runOneStep := FALSE;
        RETURN;
    END_IF
END_IF

IF SUPER^.Step(28, TRUE, 'Step number 28') THEN
    SUPER^.StepCompleteWhen((_runOneStep OR _runAllSteps) AND _finishStep);

    IF _runOneStep THEN
        _runOneStep := FALSE;
        RETURN;
    END_IF
END_IF

IF SUPER^.Step(29, TRUE, 'Step number 29') THEN
    SUPER^.StepCompleteWhen((_runOneStep OR _runAllSteps) AND _finishStep);

    IF _runOneStep THEN
        _runOneStep := FALSE;
        RETURN;
    END_IF
END_IF

IF SUPER^.Step(30, TRUE, 'Step number 30') THEN
    SUPER^.StepCompleteWhen((_runOneStep OR _runAllSteps) AND _finishStep);

    IF _runOneStep THEN
        _runOneStep := FALSE;
        RETURN;
    END_IF
END_IF

IF SUPER^.Step(31, TRUE, 'Step number 31') THEN
    SUPER^.StepCompleteWhen((_runOneStep OR _runAllSteps) AND _finishStep);

    IF _runOneStep THEN
        _runOneStep := FALSE;
        RETURN;
    END_IF
END_IF

IF SUPER^.Step(32, TRUE, 'Step number 32') THEN
    SUPER^.StepCompleteWhen((_runOneStep OR _runAllSteps) AND _finishStep);

    IF _runOneStep THEN
        _runOneStep := FALSE;
        RETURN;
    END_IF
END_IF

IF SUPER^.Step(33, TRUE, 'Step number 33') THEN
    SUPER^.StepCompleteWhen((_runOneStep OR _runAllSteps) AND _finishStep);

    IF _runOneStep THEN
        _runOneStep := FALSE;
        RETURN;
    END_IF
END_IF

IF SUPER^.Step(34, TRUE, 'Step number 34') THEN
    SUPER^.StepCompleteWhen((_runOneStep OR _runAllSteps) AND _finishStep);

    IF _runOneStep THEN
        _runOneStep := FALSE;
        RETURN;
    END_IF
END_IF

IF SUPER^.Step(35, TRUE, 'Step number 35') THEN
    SUPER^.StepCompleteWhen((_runOneStep OR _runAllSteps) AND _finishStep);

    IF _runOneStep THEN
        _runOneStep := FALSE;
        RETURN;
    END_IF
END_IF

IF SUPER^.Step(36, TRUE, 'Step number 36') THEN
    SUPER^.StepCompleteWhen((_runOneStep OR _runAllSteps) AND _finishStep);

    IF _runOneStep THEN
        _runOneStep := FALSE;
        RETURN;
    END_IF
END_IF

IF SUPER^.Step(37, TRUE, 'Step number 37') THEN
    SUPER^.StepCompleteWhen((_runOneStep OR _runAllSteps) AND _finishStep);

    IF _runOneStep THEN
        _runOneStep := FALSE;
        RETURN;
    END_IF
END_IF

IF SUPER^.Step(38, TRUE, 'Step number 38') THEN
    SUPER^.StepCompleteWhen((_runOneStep OR _runAllSteps) AND _finishStep);

    IF _runOneStep THEN
        _runOneStep := FALSE;
        RETURN;
    END_IF
END_IF

IF SUPER^.Step(39, TRUE, 'Step number 39') THEN
    SUPER^.StepCompleteWhen((_runOneStep OR _runAllSteps) AND _finishStep);

    IF _runOneStep THEN
        _runOneStep := FALSE;
        RETURN;
    END_IF
END_IF

IF SUPER^.Step(40, TRUE, 'Step number 40') THEN
    SUPER^.StepCompleteWhen((_runOneStep OR _runAllSteps) AND _finishStep);

    IF _runOneStep THEN
        _runOneStep := FALSE;
        RETURN;
    END_IF
END_IF

IF SUPER^.Step(41, TRUE, 'Step number 41') THEN
    SUPER^.StepCompleteWhen((_runOneStep OR _runAllSteps) AND _finishStep);

    IF _runOneStep THEN
        _runOneStep := FALSE;
        RETURN;
    END_IF
END_IF

IF SUPER^.Step(42, TRUE, 'Step number 42') THEN
    SUPER^.StepCompleteWhen((_runOneStep OR _runAllSteps) AND _finishStep);

    IF _runOneStep THEN
        _runOneStep := FALSE;
        RETURN;
    END_IF
END_IF

IF SUPER^.Step(43, TRUE, 'Step number 43') THEN
    SUPER^.StepCompleteWhen((_runOneStep OR _runAllSteps) AND _finishStep);

    IF _runOneStep THEN
        _runOneStep := FALSE;
        RETURN;
    END_IF
END_IF

IF SUPER^.Step(44, TRUE, 'Step number 44') THEN
    SUPER^.StepCompleteWhen((_runOneStep OR _runAllSteps) AND _finishStep);

    IF _runOneStep THEN
        _runOneStep := FALSE;
        RETURN;
    END_IF
END_IF

IF SUPER^.Step(45, TRUE, 'Step number 45') THEN
    SUPER^.StepCompleteWhen((_runOneStep OR _runAllSteps) AND _finishStep);

    IF _runOneStep THEN
        _runOneStep := FALSE;
        RETURN;
    END_IF
END_IF

IF SUPER^.Step(46, TRUE, 'Step number 46') THEN
    SUPER^.StepCompleteWhen((_runOneStep OR _runAllSteps) AND _finishStep);

    IF _runOneStep THEN
        _runOneStep := FALSE;
        RETURN;
    END_IF
END_IF

IF SUPER^.Step(47, TRUE, 'Step number 47') THEN
    SUPER^.StepCompleteWhen((_runOneStep OR _runAllSteps) AND _finishStep);

    IF _runOneStep THEN
        _runOneStep := FALSE;
        RETURN;
    END_IF
END_IF

IF SUPER^.Step(48, TRUE, 'Step number 48') THEN
    SUPER^.StepCompleteWhen((_runOneStep OR _runAllSteps) AND _finishStep);

    IF _runOneStep THEN
        _runOneStep := FALSE;
        RETURN;
    END_IF
END_IF

IF SUPER^.Step(49, TRUE, 'Step number 49') THEN
    SUPER^.StepCompleteWhen((_runOneStep OR _runAllSteps) AND _finishStep);

    IF _runOneStep THEN
        _runOneStep := FALSE;
        RETURN;
    END_IF
END_IF

IF SUPER^.Step(50, TRUE, 'Step number 50') THEN
    SUPER^.StepCompleteWhen((_runOneStep OR _runAllSteps) AND _finishStep);

    IF _runOneStep THEN
        _runOneStep := FALSE;
        RETURN;
    END_IF
END_IF

IF SUPER^.Step(51, TRUE, 'Step number 51') THEN
    SUPER^.StepCompleteWhen((_runOneStep OR _runAllSteps) AND _finishStep);

    IF _runOneStep THEN
        _runOneStep := FALSE;
        RETURN;
    END_IF
END_IF

IF SUPER^.Step(52, TRUE, 'Step number 52') THEN
    SUPER^.StepCompleteWhen((_runOneStep OR _runAllSteps) AND _finishStep);

    IF _runOneStep THEN
        _runOneStep := FALSE;
        RETURN;
    END_IF
END_IF

IF SUPER^.Step(53, TRUE, 'Step number 53') THEN
    SUPER^.StepCompleteWhen((_runOneStep OR _runAllSteps) AND _finishStep);

    IF _runOneStep THEN
        _runOneStep := FALSE;
        RETURN;
    END_IF
END_IF

IF SUPER^.Step(54, TRUE, 'Step number 54') THEN
    SUPER^.StepCompleteWhen((_runOneStep OR _runAllSteps) AND _finishStep);

    IF _runOneStep THEN
        _runOneStep := FALSE;
        RETURN;
    END_IF
END_IF

IF SUPER^.Step(55, TRUE, 'Step number 55') THEN
    SUPER^.StepCompleteWhen((_runOneStep OR _runAllSteps) AND _finishStep);

    IF _runOneStep THEN
        _runOneStep := FALSE;
        RETURN;
    END_IF
END_IF

IF SUPER^.Step(56, TRUE, 'Step number 56') THEN
    SUPER^.StepCompleteWhen((_runOneStep OR _runAllSteps) AND _finishStep);

    IF _runOneStep THEN
        _runOneStep := FALSE;
        RETURN;
    END_IF
END_IF

IF SUPER^.Step(57, TRUE, 'Step number 57') THEN
    SUPER^.StepCompleteWhen((_runOneStep OR _runAllSteps) AND _finishStep);

    IF _runOneStep THEN
        _runOneStep := FALSE;
        RETURN;
    END_IF
END_IF

IF SUPER^.Step(58, TRUE, 'Step number 58') THEN
    SUPER^.StepCompleteWhen((_runOneStep OR _runAllSteps) AND _finishStep);

    IF _runOneStep THEN
        _runOneStep := FALSE;
        RETURN;
    END_IF
END_IF

IF SUPER^.Step(59, TRUE, 'Step number 59') THEN
    SUPER^.StepCompleteWhen((_runOneStep OR _runAllSteps) AND _finishStep);

    IF _runOneStep THEN
        _runOneStep := FALSE;
        RETURN;
    END_IF
END_IF

IF SUPER^.Step(60, TRUE, 'Step number 60') THEN
    SUPER^.StepCompleteWhen((_runOneStep OR _runAllSteps) AND _finishStep);

    IF _runOneStep THEN
        _runOneStep := FALSE;
        RETURN;
    END_IF
END_IF

IF SUPER^.Step(61, TRUE, 'Step number 61') THEN
    SUPER^.StepCompleteWhen((_runOneStep OR _runAllSteps) AND _finishStep);

    IF _runOneStep THEN
        _runOneStep := FALSE;
        RETURN;
    END_IF
END_IF

IF SUPER^.Step(62, TRUE, 'Step number 62') THEN
    SUPER^.StepCompleteWhen((_runOneStep OR _runAllSteps) AND _finishStep);

    IF _runOneStep THEN
        _runOneStep := FALSE;
        RETURN;
    END_IF
END_IF

IF SUPER^.Step(63, TRUE, 'Step number 63') THEN
    SUPER^.StepCompleteWhen((_runOneStep OR _runAllSteps) AND _finishStep);

    IF _runOneStep THEN
        _runOneStep := FALSE;
        RETURN;
    END_IF
END_IF

IF SUPER^.Step(64, TRUE, 'Step number 64') THEN
    SUPER^.StepCompleteWhen((_runOneStep OR _runAllSteps) AND _finishStep);

    IF _runOneStep THEN
        _runOneStep := FALSE;
        RETURN;
    END_IF
END_IF

IF SUPER^.Step(65, TRUE, 'Step number 65') THEN
    SUPER^.StepCompleteWhen((_runOneStep OR _runAllSteps) AND _finishStep);

    IF _runOneStep THEN
        _runOneStep := FALSE;
        RETURN;
    END_IF
END_IF

IF SUPER^.Step(66, TRUE, 'Step number 66') THEN
    SUPER^.StepCompleteWhen((_runOneStep OR _runAllSteps) AND _finishStep);

    IF _runOneStep THEN
        _runOneStep := FALSE;
        RETURN;
    END_IF
END_IF

IF SUPER^.Step(67, TRUE, 'Step number 67') THEN
    SUPER^.StepCompleteWhen((_runOneStep OR _runAllSteps) AND _finishStep);

    IF _runOneStep THEN
        _runOneStep := FALSE;
        RETURN;
    END_IF
END_IF

IF SUPER^.Step(68, TRUE, 'Step number 68') THEN
    SUPER^.StepCompleteWhen((_runOneStep OR _runAllSteps) AND _finishStep);

    IF _runOneStep THEN
        _runOneStep := FALSE;
        RETURN;
    END_IF
END_IF

IF SUPER^.Step(69, TRUE, 'Step number 69') THEN
    SUPER^.StepCompleteWhen((_runOneStep OR _runAllSteps) AND _finishStep);

    IF _runOneStep THEN
        _runOneStep := FALSE;
        RETURN;
    END_IF
END_IF

IF SUPER^.Step(70, TRUE, 'Step number 70') THEN
    SUPER^.StepCompleteWhen((_runOneStep OR _runAllSteps) AND _finishStep);

    IF _runOneStep THEN
        _runOneStep := FALSE;
        RETURN;
    END_IF
END_IF

IF SUPER^.Step(71, TRUE, 'Step number 71') THEN
    SUPER^.StepCompleteWhen((_runOneStep OR _runAllSteps) AND _finishStep);

    IF _runOneStep THEN
        _runOneStep := FALSE;
        RETURN;
    END_IF
END_IF

IF SUPER^.Step(72, TRUE, 'Step number 72') THEN
    SUPER^.StepCompleteWhen((_runOneStep OR _runAllSteps) AND _finishStep);

    IF _runOneStep THEN
        _runOneStep := FALSE;
        RETURN;
    END_IF
END_IF

IF SUPER^.Step(73, TRUE, 'Step number 73') THEN
    SUPER^.StepCompleteWhen((_runOneStep OR _runAllSteps) AND _finishStep);

    IF _runOneStep THEN
        _runOneStep := FALSE;
        RETURN;
    END_IF
END_IF

IF SUPER^.Step(74, TRUE, 'Step number 74') THEN
    SUPER^.StepCompleteWhen((_runOneStep OR _runAllSteps) AND _finishStep);

    IF _runOneStep THEN
        _runOneStep := FALSE;
        RETURN;
    END_IF
END_IF

IF SUPER^.Step(75, TRUE, 'Step number 75') THEN
    SUPER^.StepCompleteWhen((_runOneStep OR _runAllSteps) AND _finishStep);

    IF _runOneStep THEN
        _runOneStep := FALSE;
        RETURN;
    END_IF
END_IF

IF SUPER^.Step(76, TRUE, 'Step number 76') THEN
    SUPER^.StepCompleteWhen((_runOneStep OR _runAllSteps) AND _finishStep);

    IF _runOneStep THEN
        _runOneStep := FALSE;
        RETURN;
    END_IF
END_IF

IF SUPER^.Step(77, TRUE, 'Step number 77') THEN
    SUPER^.StepCompleteWhen((_runOneStep OR _runAllSteps) AND _finishStep);

    IF _runOneStep THEN
        _runOneStep := FALSE;
        RETURN;
    END_IF
END_IF

IF SUPER^.Step(78, TRUE, 'Step number 78') THEN
    SUPER^.StepCompleteWhen((_runOneStep OR _runAllSteps) AND _finishStep);

    IF _runOneStep THEN
        _runOneStep := FALSE;
        RETURN;
    END_IF
END_IF

IF SUPER^.Step(79, TRUE, 'Step number 79') THEN
    SUPER^.StepCompleteWhen((_runOneStep OR _runAllSteps) AND _finishStep);

    IF _runOneStep THEN
        _runOneStep := FALSE;
        RETURN;
    END_IF
END_IF

IF SUPER^.Step(80, TRUE, 'Step number 80') THEN
    SUPER^.StepCompleteWhen((_runOneStep OR _runAllSteps) AND _finishStep);

    IF _runOneStep THEN
        _runOneStep := FALSE;
        RETURN;
    END_IF
END_IF

IF SUPER^.Step(81, TRUE, 'Step number 81') THEN
    SUPER^.StepCompleteWhen((_runOneStep OR _runAllSteps) AND _finishStep);

    IF _runOneStep THEN
        _runOneStep := FALSE;
        RETURN;
    END_IF
END_IF

IF SUPER^.Step(82, TRUE, 'Step number 82') THEN
    SUPER^.StepCompleteWhen((_runOneStep OR _runAllSteps) AND _finishStep);

    IF _runOneStep THEN
        _runOneStep := FALSE;
        RETURN;
    END_IF
END_IF

IF SUPER^.Step(83, TRUE, 'Step number 83') THEN
    SUPER^.StepCompleteWhen((_runOneStep OR _runAllSteps) AND _finishStep);

    IF _runOneStep THEN
        _runOneStep := FALSE;
        RETURN;
    END_IF
END_IF

IF SUPER^.Step(84, TRUE, 'Step number 84') THEN
    SUPER^.StepCompleteWhen((_runOneStep OR _runAllSteps) AND _finishStep);

    IF _runOneStep THEN
        _runOneStep := FALSE;
        RETURN;
    END_IF
END_IF

IF SUPER^.Step(85, TRUE, 'Step number 85') THEN
    SUPER^.StepCompleteWhen((_runOneStep OR _runAllSteps) AND _finishStep);

    IF _runOneStep THEN
        _runOneStep := FALSE;
        RETURN;
    END_IF
END_IF

IF SUPER^.Step(86, TRUE, 'Step number 86') THEN
    SUPER^.StepCompleteWhen((_runOneStep OR _runAllSteps) AND _finishStep);

    IF _runOneStep THEN
        _runOneStep := FALSE;
        RETURN;
    END_IF
END_IF

IF SUPER^.Step(87, TRUE, 'Step number 87') THEN
    SUPER^.StepCompleteWhen((_runOneStep OR _runAllSteps) AND _finishStep);

    IF _runOneStep THEN
        _runOneStep := FALSE;
        RETURN;
    END_IF
END_IF

IF SUPER^.Step(88, TRUE, 'Step number 88') THEN
    SUPER^.StepCompleteWhen((_runOneStep OR _runAllSteps) AND _finishStep);

    IF _runOneStep THEN
        _runOneStep := FALSE;
        RETURN;
    END_IF
END_IF

IF SUPER^.Step(89, TRUE, 'Step number 89') THEN
    SUPER^.StepCompleteWhen((_runOneStep OR _runAllSteps) AND _finishStep);

    IF _runOneStep THEN
        _runOneStep := FALSE;
        RETURN;
    END_IF
END_IF

IF SUPER^.Step(90, TRUE, 'Step number 90') THEN
    SUPER^.StepCompleteWhen((_runOneStep OR _runAllSteps) AND _finishStep);

    IF _runOneStep THEN
        _runOneStep := FALSE;
        RETURN;
    END_IF
END_IF

IF SUPER^.Step(91, TRUE, 'Step number 91') THEN
    SUPER^.StepCompleteWhen((_runOneStep OR _runAllSteps) AND _finishStep);

    IF _runOneStep THEN
        _runOneStep := FALSE;
        RETURN;
    END_IF
END_IF

IF SUPER^.Step(92, TRUE, 'Step number 92') THEN
    SUPER^.StepCompleteWhen((_runOneStep OR _runAllSteps) AND _finishStep);

    IF _runOneStep THEN
        _runOneStep := FALSE;
        RETURN;
    END_IF
END_IF

IF SUPER^.Step(93, TRUE, 'Step number 93') THEN
    SUPER^.StepCompleteWhen((_runOneStep OR _runAllSteps) AND _finishStep);

    IF _runOneStep THEN
        _runOneStep := FALSE;
        RETURN;
    END_IF
END_IF

IF SUPER^.Step(94, TRUE, 'Step number 94') THEN
    SUPER^.StepCompleteWhen((_runOneStep OR _runAllSteps) AND _finishStep);

    IF _runOneStep THEN
        _runOneStep := FALSE;
        RETURN;
    END_IF
END_IF

IF SUPER^.Step(95, TRUE, 'Step number 95') THEN
    SUPER^.StepCompleteWhen((_runOneStep OR _runAllSteps) AND _finishStep);

    IF _runOneStep THEN
        _runOneStep := FALSE;
        RETURN;
    END_IF
END_IF

IF SUPER^.Step(96, TRUE, 'Step number 96') THEN
    SUPER^.StepCompleteWhen((_runOneStep OR _runAllSteps) AND _finishStep);

    IF _runOneStep THEN
        _runOneStep := FALSE;
        RETURN;
    END_IF
END_IF

IF SUPER^.Step(97, TRUE, 'Step number 97') THEN
    SUPER^.StepCompleteWhen((_runOneStep OR _runAllSteps) AND _finishStep);

    IF _runOneStep THEN
        _runOneStep := FALSE;
        RETURN;
    END_IF
END_IF

IF SUPER^.Step(98, TRUE, 'Step number 98') THEN
    SUPER^.StepCompleteWhen((_runOneStep OR _runAllSteps) AND _finishStep);

    IF _runOneStep THEN
        _runOneStep := FALSE;
        RETURN;
    END_IF
END_IF

IF SUPER^.Step(99, TRUE, 'Step number 99') THEN
    SUPER^.StepCompleteWhen((_runOneStep OR _runAllSteps) AND _finishStep);

    IF _runOneStep THEN
        _runOneStep := FALSE;
        RETURN;
    END_IF
END_IF

IF SUPER^.Step(100, TRUE, 'Step number 100') THEN
    SUPER^.StepCompleteWhen((_runOneStep OR _runAllSteps) AND _finishStep);

    IF _runOneStep THEN
        _runOneStep := FALSE;
        RETURN;
    END_IF
END_IF

IF SUPER^.Step(101, TRUE, 'Step number 101') THEN
    SUPER^.StepCompleteWhen((_runOneStep OR _runAllSteps) AND _finishStep);

    IF _runOneStep THEN
        _runOneStep := FALSE;
        RETURN;
    END_IF
END_IF

IF SUPER^.Step(102, TRUE, 'Step number 102') THEN
    SUPER^.StepCompleteWhen((_runOneStep OR _runAllSteps) AND _finishStep);

    IF _runOneStep THEN
        _runOneStep := FALSE;
        RETURN;
    END_IF
END_IF

IF SUPER^.Step(103, TRUE, 'Step number 103') THEN
    SUPER^.StepCompleteWhen((_runOneStep OR _runAllSteps) AND _finishStep);

    IF _runOneStep THEN
        _runOneStep := FALSE;
        RETURN;
    END_IF
END_IF

IF SUPER^.Step(104, TRUE, 'Step number 104') THEN
    SUPER^.StepCompleteWhen((_runOneStep OR _runAllSteps) AND _finishStep);

    IF _runOneStep THEN
        _runOneStep := FALSE;
        RETURN;
    END_IF
END_IF

IF SUPER^.Step(105, TRUE, 'Step number 105') THEN
    SUPER^.StepCompleteWhen((_runOneStep OR _runAllSteps) AND _finishStep);

    IF _runOneStep THEN
        _runOneStep := FALSE;
        RETURN;
    END_IF
END_IF

IF SUPER^.Step(106, TRUE, 'Step number 106') THEN
    SUPER^.StepCompleteWhen((_runOneStep OR _runAllSteps) AND _finishStep);

    IF _runOneStep THEN
        _runOneStep := FALSE;
        RETURN;
    END_IF
END_IF

IF SUPER^.Step(107, TRUE, 'Step number 107') THEN
    SUPER^.StepCompleteWhen((_runOneStep OR _runAllSteps) AND _finishStep);

    IF _runOneStep THEN
        _runOneStep := FALSE;
        RETURN;
    END_IF
END_IF

IF SUPER^.Step(108, TRUE, 'Step number 108') THEN
    SUPER^.StepCompleteWhen((_runOneStep OR _runAllSteps) AND _finishStep);

    IF _runOneStep THEN
        _runOneStep := FALSE;
        RETURN;
    END_IF
END_IF

IF SUPER^.Step(109, TRUE, 'Step number 109') THEN
    SUPER^.StepCompleteWhen((_runOneStep OR _runAllSteps) AND _finishStep);

    IF _runOneStep THEN
        _runOneStep := FALSE;
        RETURN;
    END_IF
END_IF

IF SUPER^.Step(110, TRUE, 'Step number 110') THEN
    SUPER^.StepCompleteWhen((_runOneStep OR _runAllSteps) AND _finishStep);

    IF _runOneStep THEN
        _runOneStep := FALSE;
        RETURN;
    END_IF
END_IF

IF SUPER^.Step(111, TRUE, 'Step number 111') THEN
    SUPER^.StepCompleteWhen((_runOneStep OR _runAllSteps) AND _finishStep);

    IF _runOneStep THEN
        _runOneStep := FALSE;
        RETURN;
    END_IF
END_IF

IF SUPER^.Step(112, TRUE, 'Step number 112') THEN
    SUPER^.StepCompleteWhen((_runOneStep OR _runAllSteps) AND _finishStep);

    IF _runOneStep THEN
        _runOneStep := FALSE;
        RETURN;
    END_IF
END_IF

IF SUPER^.Step(113, TRUE, 'Step number 113') THEN
    SUPER^.StepCompleteWhen((_runOneStep OR _runAllSteps) AND _finishStep);

    IF _runOneStep THEN
        _runOneStep := FALSE;
        RETURN;
    END_IF
END_IF

IF SUPER^.Step(114, TRUE, 'Step number 114') THEN
    SUPER^.StepCompleteWhen((_runOneStep OR _runAllSteps) AND _finishStep);

    IF _runOneStep THEN
        _runOneStep := FALSE;
        RETURN;
    END_IF
END_IF

IF SUPER^.Step(115, TRUE, 'Step number 115') THEN
    SUPER^.StepCompleteWhen((_runOneStep OR _runAllSteps) AND _finishStep);

    IF _runOneStep THEN
        _runOneStep := FALSE;
        RETURN;
    END_IF
END_IF

IF SUPER^.Step(116, TRUE, 'Step number 116') THEN
    SUPER^.StepCompleteWhen((_runOneStep OR _runAllSteps) AND _finishStep);

    IF _runOneStep THEN
        _runOneStep := FALSE;
        RETURN;
    END_IF
END_IF

IF SUPER^.Step(117, TRUE, 'Step number 117') THEN
    SUPER^.StepCompleteWhen((_runOneStep OR _runAllSteps) AND _finishStep);

    IF _runOneStep THEN
        _runOneStep := FALSE;
        RETURN;
    END_IF
END_IF

IF SUPER^.Step(118, TRUE, 'Step number 118') THEN
    SUPER^.StepCompleteWhen((_runOneStep OR _runAllSteps) AND _finishStep);

    IF _runOneStep THEN
        _runOneStep := FALSE;
        RETURN;
    END_IF
END_IF

IF SUPER^.Step(119, TRUE, 'Step number 119') THEN
    SUPER^.StepCompleteWhen((_runOneStep OR _runAllSteps) AND _finishStep);

    IF _runOneStep THEN
        _runOneStep := FALSE;
        RETURN;
    END_IF
END_IF

IF SUPER^.Step(120, TRUE, 'Step number 120') THEN
    SUPER^.StepCompleteWhen((_runOneStep OR _runAllSteps) AND _finishStep);

    IF _runOneStep THEN
        _runOneStep := FALSE;
        RETURN;
    END_IF
END_IF

IF SUPER^.Step(121, TRUE, 'Step number 121') THEN
    SUPER^.StepCompleteWhen((_runOneStep OR _runAllSteps) AND _finishStep);

    IF _runOneStep THEN
        _runOneStep := FALSE;
        RETURN;
    END_IF
END_IF

IF SUPER^.Step(122, TRUE, 'Step number 122') THEN
    SUPER^.StepCompleteWhen((_runOneStep OR _runAllSteps) AND _finishStep);

    IF _runOneStep THEN
        _runOneStep := FALSE;
        RETURN;
    END_IF
END_IF

IF SUPER^.Step(123, TRUE, 'Step number 123') THEN
    SUPER^.StepCompleteWhen((_runOneStep OR _runAllSteps) AND _finishStep);

    IF _runOneStep THEN
        _runOneStep := FALSE;
        RETURN;
    END_IF
END_IF

IF SUPER^.Step(124, TRUE, 'Step number 124') THEN
    SUPER^.StepCompleteWhen((_runOneStep OR _runAllSteps) AND _finishStep);

    IF _runOneStep THEN
        _runOneStep := FALSE;
        RETURN;
    END_IF
END_IF

IF SUPER^.Step(125, TRUE, 'Step number 125') THEN
    SUPER^.StepCompleteWhen((_runOneStep OR _runAllSteps) AND _finishStep);

    IF _runOneStep THEN
        _runOneStep := FALSE;
        RETURN;
    END_IF
END_IF

IF SUPER^.Step(126, TRUE, 'Step number 126') THEN
    SUPER^.StepCompleteWhen((_runOneStep OR _runAllSteps) AND _finishStep);

    IF _runOneStep THEN
        _runOneStep := FALSE;
        RETURN;
    END_IF
END_IF

IF SUPER^.Step(127, TRUE, 'Step number 127') THEN
    SUPER^.StepCompleteWhen((_runOneStep OR _runAllSteps) AND _finishStep);

    IF _runOneStep THEN
        _runOneStep := FALSE;
        RETURN;
    END_IF
END_IF

IF SUPER^.Step(128, TRUE, 'Step number 128') THEN
    SUPER^.StepCompleteWhen((_runOneStep OR _runAllSteps) AND _finishStep);

    IF _runOneStep THEN
        _runOneStep := FALSE;
        RETURN;
    END_IF
END_IF

IF SUPER^.Step(129, TRUE, 'Step number 129') THEN
    SUPER^.StepCompleteWhen((_runOneStep OR _runAllSteps) AND _finishStep);

    IF _runOneStep THEN
        _runOneStep := FALSE;
        RETURN;
    END_IF
END_IF

IF SUPER^.Step(130, TRUE, 'Step number 130') THEN
    SUPER^.StepCompleteWhen((_runOneStep OR _runAllSteps) AND _finishStep);

    IF _runOneStep THEN
        _runOneStep := FALSE;
        RETURN;
    END_IF
END_IF

IF SUPER^.Step(131, TRUE, 'Step number 131') THEN
    SUPER^.StepCompleteWhen((_runOneStep OR _runAllSteps) AND _finishStep);

    IF _runOneStep THEN
        _runOneStep := FALSE;
        RETURN;
    END_IF
END_IF

IF SUPER^.Step(132, TRUE, 'Step number 132') THEN
    SUPER^.StepCompleteWhen((_runOneStep OR _runAllSteps) AND _finishStep);

    IF _runOneStep THEN
        _runOneStep := FALSE;
        RETURN;
    END_IF
END_IF

IF SUPER^.Step(133, TRUE, 'Step number 133') THEN
    SUPER^.StepCompleteWhen((_runOneStep OR _runAllSteps) AND _finishStep);

    IF _runOneStep THEN
        _runOneStep := FALSE;
        RETURN;
    END_IF
END_IF

IF SUPER^.Step(134, TRUE, 'Step number 134') THEN
    SUPER^.StepCompleteWhen((_runOneStep OR _runAllSteps) AND _finishStep);

    IF _runOneStep THEN
        _runOneStep := FALSE;
        RETURN;
    END_IF
END_IF

IF SUPER^.Step(135, TRUE, 'Step number 135') THEN
    SUPER^.StepCompleteWhen((_runOneStep OR _runAllSteps) AND _finishStep);

    IF _runOneStep THEN
        _runOneStep := FALSE;
        RETURN;
    END_IF
END_IF

IF SUPER^.Step(136, TRUE, 'Step number 136') THEN
    SUPER^.StepCompleteWhen((_runOneStep OR _runAllSteps) AND _finishStep);

    IF _runOneStep THEN
        _runOneStep := FALSE;
        RETURN;
    END_IF
END_IF

IF SUPER^.Step(137, TRUE, 'Step number 137') THEN
    SUPER^.StepCompleteWhen((_runOneStep OR _runAllSteps) AND _finishStep);

    IF _runOneStep THEN
        _runOneStep := FALSE;
        RETURN;
    END_IF
END_IF

IF SUPER^.Step(138, TRUE, 'Step number 138') THEN
    SUPER^.StepCompleteWhen((_runOneStep OR _runAllSteps) AND _finishStep);

    IF _runOneStep THEN
        _runOneStep := FALSE;
        RETURN;
    END_IF
END_IF

IF SUPER^.Step(139, TRUE, 'Step number 139') THEN
    SUPER^.StepCompleteWhen((_runOneStep OR _runAllSteps) AND _finishStep);

    IF _runOneStep THEN
        _runOneStep := FALSE;
        RETURN;
    END_IF
END_IF

IF SUPER^.Step(140, TRUE, 'Step number 140') THEN
    SUPER^.StepCompleteWhen((_runOneStep OR _runAllSteps) AND _finishStep);

    IF _runOneStep THEN
        _runOneStep := FALSE;
        RETURN;
    END_IF
END_IF

IF SUPER^.Step(141, TRUE, 'Step number 141') THEN
    SUPER^.StepCompleteWhen((_runOneStep OR _runAllSteps) AND _finishStep);

    IF _runOneStep THEN
        _runOneStep := FALSE;
        RETURN;
    END_IF
END_IF

IF SUPER^.Step(142, TRUE, 'Step number 142') THEN
    SUPER^.StepCompleteWhen((_runOneStep OR _runAllSteps) AND _finishStep);

    IF _runOneStep THEN
        _runOneStep := FALSE;
        RETURN;
    END_IF
END_IF

IF SUPER^.Step(143, TRUE, 'Step number 143') THEN
    SUPER^.StepCompleteWhen((_runOneStep OR _runAllSteps) AND _finishStep);

    IF _runOneStep THEN
        _runOneStep := FALSE;
        RETURN;
    END_IF
END_IF

IF SUPER^.Step(144, TRUE, 'Step number 144') THEN
    SUPER^.StepCompleteWhen((_runOneStep OR _runAllSteps) AND _finishStep);

    IF _runOneStep THEN
        _runOneStep := FALSE;
        RETURN;
    END_IF
END_IF

IF SUPER^.Step(145, TRUE, 'Step number 145') THEN
    SUPER^.StepCompleteWhen((_runOneStep OR _runAllSteps) AND _finishStep);

    IF _runOneStep THEN
        _runOneStep := FALSE;
        RETURN;
    END_IF
END_IF

IF SUPER^.Step(146, TRUE, 'Step number 146') THEN
    SUPER^.StepCompleteWhen((_runOneStep OR _runAllSteps) AND _finishStep);

    IF _runOneStep THEN
        _runOneStep := FALSE;
        RETURN;
    END_IF
END_IF

IF SUPER^.Step(147, TRUE, 'Step number 147') THEN
    SUPER^.StepCompleteWhen((_runOneStep OR _runAllSteps) AND _finishStep);

    IF _runOneStep THEN
        _runOneStep := FALSE;
        RETURN;
    END_IF
END_IF

IF SUPER^.Step(148, TRUE, 'Step number 148') THEN
    SUPER^.StepCompleteWhen((_runOneStep OR _runAllSteps) AND _finishStep);

    IF _runOneStep THEN
        _runOneStep := FALSE;
        RETURN;
    END_IF
END_IF

IF SUPER^.Step(149, TRUE, 'Step number 149') THEN
    SUPER^.StepCompleteWhen((_runOneStep OR _runAllSteps) AND _finishStep);

    IF _runOneStep THEN
        _runOneStep := FALSE;
        RETURN;
    END_IF
END_IF

IF SUPER^.Step(150, TRUE, 'Step number 150') THEN
    SUPER^.StepCompleteWhen((_runOneStep OR _runAllSteps) AND _finishStep);

    IF _runOneStep THEN
        _runOneStep := FALSE;
        RETURN;
    END_IF
END_IF

IF SUPER^.Step(151, TRUE, 'Step number 151') THEN
    SUPER^.StepCompleteWhen((_runOneStep OR _runAllSteps) AND _finishStep);

    IF _runOneStep THEN
        _runOneStep := FALSE;
        RETURN;
    END_IF
END_IF

IF SUPER^.Step(152, TRUE, 'Step number 152') THEN
    SUPER^.StepCompleteWhen((_runOneStep OR _runAllSteps) AND _finishStep);

    IF _runOneStep THEN
        _runOneStep := FALSE;
        RETURN;
    END_IF
END_IF

IF SUPER^.Step(153, TRUE, 'Step number 153') THEN
    SUPER^.StepCompleteWhen((_runOneStep OR _runAllSteps) AND _finishStep);

    IF _runOneStep THEN
        _runOneStep := FALSE;
        RETURN;
    END_IF
END_IF

IF SUPER^.Step(154, TRUE, 'Step number 154') THEN
    SUPER^.StepCompleteWhen((_runOneStep OR _runAllSteps) AND _finishStep);

    IF _runOneStep THEN
        _runOneStep := FALSE;
        RETURN;
    END_IF
END_IF

IF SUPER^.Step(155, TRUE, 'Step number 155') THEN
    SUPER^.StepCompleteWhen((_runOneStep OR _runAllSteps) AND _finishStep);

    IF _runOneStep THEN
        _runOneStep := FALSE;
        RETURN;
    END_IF
END_IF

IF SUPER^.Step(156, TRUE, 'Step number 156') THEN
    SUPER^.StepCompleteWhen((_runOneStep OR _runAllSteps) AND _finishStep);

    IF _runOneStep THEN
        _runOneStep := FALSE;
        RETURN;
    END_IF
END_IF

IF SUPER^.Step(157, TRUE, 'Step number 157') THEN
    SUPER^.StepCompleteWhen((_runOneStep OR _runAllSteps) AND _finishStep);

    IF _runOneStep THEN
        _runOneStep := FALSE;
        RETURN;
    END_IF
END_IF

IF SUPER^.Step(158, TRUE, 'Step number 158') THEN
    SUPER^.StepCompleteWhen((_runOneStep OR _runAllSteps) AND _finishStep);

    IF _runOneStep THEN
        _runOneStep := FALSE;
        RETURN;
    END_IF
END_IF

IF SUPER^.Step(159, TRUE, 'Step number 159') THEN
    SUPER^.StepCompleteWhen((_runOneStep OR _runAllSteps) AND _finishStep);

    IF _runOneStep THEN
        _runOneStep := FALSE;
        RETURN;
    END_IF
END_IF

IF SUPER^.Step(160, TRUE, 'Step number 160') THEN
    SUPER^.StepCompleteWhen((_runOneStep OR _runAllSteps) AND _finishStep);

    IF _runOneStep THEN
        _runOneStep := FALSE;
        RETURN;
    END_IF
END_IF

IF SUPER^.Step(161, TRUE, 'Step number 161') THEN
    SUPER^.StepCompleteWhen((_runOneStep OR _runAllSteps) AND _finishStep);

    IF _runOneStep THEN
        _runOneStep := FALSE;
        RETURN;
    END_IF
END_IF

IF SUPER^.Step(162, TRUE, 'Step number 162') THEN
    SUPER^.StepCompleteWhen((_runOneStep OR _runAllSteps) AND _finishStep);

    IF _runOneStep THEN
        _runOneStep := FALSE;
        RETURN;
    END_IF
END_IF

IF SUPER^.Step(163, TRUE, 'Step number 163') THEN
    SUPER^.StepCompleteWhen((_runOneStep OR _runAllSteps) AND _finishStep);

    IF _runOneStep THEN
        _runOneStep := FALSE;
        RETURN;
    END_IF
END_IF

IF SUPER^.Step(164, TRUE, 'Step number 164') THEN
    SUPER^.StepCompleteWhen((_runOneStep OR _runAllSteps) AND _finishStep);

    IF _runOneStep THEN
        _runOneStep := FALSE;
        RETURN;
    END_IF
END_IF

IF SUPER^.Step(165, TRUE, 'Step number 165') THEN
    SUPER^.StepCompleteWhen((_runOneStep OR _runAllSteps) AND _finishStep);

    IF _runOneStep THEN
        _runOneStep := FALSE;
        RETURN;
    END_IF
END_IF

IF SUPER^.Step(166, TRUE, 'Step number 166') THEN
    SUPER^.StepCompleteWhen((_runOneStep OR _runAllSteps) AND _finishStep);

    IF _runOneStep THEN
        _runOneStep := FALSE;
        RETURN;
    END_IF
END_IF

IF SUPER^.Step(167, TRUE, 'Step number 167') THEN
    SUPER^.StepCompleteWhen((_runOneStep OR _runAllSteps) AND _finishStep);

    IF _runOneStep THEN
        _runOneStep := FALSE;
        RETURN;
    END_IF
END_IF

IF SUPER^.Step(168, TRUE, 'Step number 168') THEN
    SUPER^.StepCompleteWhen((_runOneStep OR _runAllSteps) AND _finishStep);

    IF _runOneStep THEN
        _runOneStep := FALSE;
        RETURN;
    END_IF
END_IF

IF SUPER^.Step(169, TRUE, 'Step number 169') THEN
    SUPER^.StepCompleteWhen((_runOneStep OR _runAllSteps) AND _finishStep);

    IF _runOneStep THEN
        _runOneStep := FALSE;
        RETURN;
    END_IF
END_IF

IF SUPER^.Step(170, TRUE, 'Step number 170') THEN
    SUPER^.StepCompleteWhen((_runOneStep OR _runAllSteps) AND _finishStep);

    IF _runOneStep THEN
        _runOneStep := FALSE;
        RETURN;
    END_IF
END_IF

IF SUPER^.Step(171, TRUE, 'Step number 171') THEN
    SUPER^.StepCompleteWhen((_runOneStep OR _runAllSteps) AND _finishStep);

    IF _runOneStep THEN
        _runOneStep := FALSE;
        RETURN;
    END_IF
END_IF

IF SUPER^.Step(172, TRUE, 'Step number 172') THEN
    SUPER^.StepCompleteWhen((_runOneStep OR _runAllSteps) AND _finishStep);

    IF _runOneStep THEN
        _runOneStep := FALSE;
        RETURN;
    END_IF
END_IF

IF SUPER^.Step(173, TRUE, 'Step number 173') THEN
    SUPER^.StepCompleteWhen((_runOneStep OR _runAllSteps) AND _finishStep);

    IF _runOneStep THEN
        _runOneStep := FALSE;
        RETURN;
    END_IF
END_IF

IF SUPER^.Step(174, TRUE, 'Step number 174') THEN
    SUPER^.StepCompleteWhen((_runOneStep OR _runAllSteps) AND _finishStep);

    IF _runOneStep THEN
        _runOneStep := FALSE;
        RETURN;
    END_IF
END_IF

IF SUPER^.Step(175, TRUE, 'Step number 175') THEN
    SUPER^.StepCompleteWhen((_runOneStep OR _runAllSteps) AND _finishStep);

    IF _runOneStep THEN
        _runOneStep := FALSE;
        RETURN;
    END_IF
END_IF

IF SUPER^.Step(176, TRUE, 'Step number 176') THEN
    SUPER^.StepCompleteWhen((_runOneStep OR _runAllSteps) AND _finishStep);

    IF _runOneStep THEN
        _runOneStep := FALSE;
        RETURN;
    END_IF
END_IF

IF SUPER^.Step(177, TRUE, 'Step number 177') THEN
    SUPER^.StepCompleteWhen((_runOneStep OR _runAllSteps) AND _finishStep);

    IF _runOneStep THEN
        _runOneStep := FALSE;
        RETURN;
    END_IF
END_IF

IF SUPER^.Step(178, TRUE, 'Step number 178') THEN
    SUPER^.StepCompleteWhen((_runOneStep OR _runAllSteps) AND _finishStep);

    IF _runOneStep THEN
        _runOneStep := FALSE;
        RETURN;
    END_IF
END_IF

IF SUPER^.Step(179, TRUE, 'Step number 179') THEN
    SUPER^.StepCompleteWhen((_runOneStep OR _runAllSteps) AND _finishStep);

    IF _runOneStep THEN
        _runOneStep := FALSE;
        RETURN;
    END_IF
END_IF

IF SUPER^.Step(180, TRUE, 'Step number 180') THEN
    SUPER^.StepCompleteWhen((_runOneStep OR _runAllSteps) AND _finishStep);

    IF _runOneStep THEN
        _runOneStep := FALSE;
        RETURN;
    END_IF
END_IF

IF SUPER^.Step(181, TRUE, 'Step number 181') THEN
    SUPER^.StepCompleteWhen((_runOneStep OR _runAllSteps) AND _finishStep);

    IF _runOneStep THEN
        _runOneStep := FALSE;
        RETURN;
    END_IF
END_IF

IF SUPER^.Step(182, TRUE, 'Step number 182') THEN
    SUPER^.StepCompleteWhen((_runOneStep OR _runAllSteps) AND _finishStep);

    IF _runOneStep THEN
        _runOneStep := FALSE;
        RETURN;
    END_IF
END_IF

IF SUPER^.Step(183, TRUE, 'Step number 183') THEN
    SUPER^.StepCompleteWhen((_runOneStep OR _runAllSteps) AND _finishStep);

    IF _runOneStep THEN
        _runOneStep := FALSE;
        RETURN;
    END_IF
END_IF

IF SUPER^.Step(184, TRUE, 'Step number 184') THEN
    SUPER^.StepCompleteWhen((_runOneStep OR _runAllSteps) AND _finishStep);

    IF _runOneStep THEN
        _runOneStep := FALSE;
        RETURN;
    END_IF
END_IF

IF SUPER^.Step(185, TRUE, 'Step number 185') THEN
    SUPER^.StepCompleteWhen((_runOneStep OR _runAllSteps) AND _finishStep);

    IF _runOneStep THEN
        _runOneStep := FALSE;
        RETURN;
    END_IF
END_IF

IF SUPER^.Step(186, TRUE, 'Step number 186') THEN
    SUPER^.StepCompleteWhen((_runOneStep OR _runAllSteps) AND _finishStep);

    IF _runOneStep THEN
        _runOneStep := FALSE;
        RETURN;
    END_IF
END_IF

IF SUPER^.Step(187, TRUE, 'Step number 187') THEN
    SUPER^.StepCompleteWhen((_runOneStep OR _runAllSteps) AND _finishStep);

    IF _runOneStep THEN
        _runOneStep := FALSE;
        RETURN;
    END_IF
END_IF

IF SUPER^.Step(188, TRUE, 'Step number 188') THEN
    SUPER^.StepCompleteWhen((_runOneStep OR _runAllSteps) AND _finishStep);

    IF _runOneStep THEN
        _runOneStep := FALSE;
        RETURN;
    END_IF
END_IF

IF SUPER^.Step(189, TRUE, 'Step number 189') THEN
    SUPER^.StepCompleteWhen((_runOneStep OR _runAllSteps) AND _finishStep);

    IF _runOneStep THEN
        _runOneStep := FALSE;
        RETURN;
    END_IF
END_IF

IF SUPER^.Step(190, TRUE, 'Step number 190') THEN
    SUPER^.StepCompleteWhen((_runOneStep OR _runAllSteps) AND _finishStep);

    IF _runOneStep THEN
        _runOneStep := FALSE;
        RETURN;
    END_IF
END_IF

IF SUPER^.Step(191, TRUE, 'Step number 191') THEN
    SUPER^.StepCompleteWhen((_runOneStep OR _runAllSteps) AND _finishStep);

    IF _runOneStep THEN
        _runOneStep := FALSE;
        RETURN;
    END_IF
END_IF

IF SUPER^.Step(192, TRUE, 'Step number 192') THEN
    SUPER^.StepCompleteWhen((_runOneStep OR _runAllSteps) AND _finishStep);

    IF _runOneStep THEN
        _runOneStep := FALSE;
        RETURN;
    END_IF
END_IF

IF SUPER^.Step(193, TRUE, 'Step number 193') THEN
    SUPER^.StepCompleteWhen((_runOneStep OR _runAllSteps) AND _finishStep);

    IF _runOneStep THEN
        _runOneStep := FALSE;
        RETURN;
    END_IF
END_IF

IF SUPER^.Step(194, TRUE, 'Step number 194') THEN
    SUPER^.StepCompleteWhen((_runOneStep OR _runAllSteps) AND _finishStep);

    IF _runOneStep THEN
        _runOneStep := FALSE;
        RETURN;
    END_IF
END_IF

IF SUPER^.Step(195, TRUE, 'Step number 195') THEN
    SUPER^.StepCompleteWhen((_runOneStep OR _runAllSteps) AND _finishStep);

    IF _runOneStep THEN
        _runOneStep := FALSE;
        RETURN;
    END_IF
END_IF

IF SUPER^.Step(196, TRUE, 'Step number 196') THEN
    SUPER^.StepCompleteWhen((_runOneStep OR _runAllSteps) AND _finishStep);

    IF _runOneStep THEN
        _runOneStep := FALSE;
        RETURN;
    END_IF
END_IF

IF SUPER^.Step(197, TRUE, 'Step number 197') THEN
    SUPER^.StepCompleteWhen((_runOneStep OR _runAllSteps) AND _finishStep);

    IF _runOneStep THEN
        _runOneStep := FALSE;
        RETURN;
    END_IF
END_IF

IF SUPER^.Step(198, TRUE, 'Step number 198') THEN
    SUPER^.StepCompleteWhen((_runOneStep OR _runAllSteps) AND _finishStep);

    IF _runOneStep THEN
        _runOneStep := FALSE;
        RETURN;
    END_IF
END_IF

IF SUPER^.Step(199, TRUE, 'Step number 199') THEN
    SUPER^.StepCompleteWhen((_runOneStep OR _runAllSteps) AND _finishStep);

    IF _runOneStep THEN
        _runOneStep := FALSE;
        RETURN;
    END_IF
END_IF

IF SUPER^.Step(200, TRUE, 'Step number 200') THEN
    SUPER^.StepCompleteWhen((_runOneStep OR _runAllSteps) AND _finishStep);

    IF _runOneStep THEN
        _runOneStep := FALSE;
        RETURN;
    END_IF
END_IF

IF SUPER^.Step(201, TRUE, 'Step number 201') THEN
    SUPER^.StepCompleteWhen((_runOneStep OR _runAllSteps) AND _finishStep);

    IF _runOneStep THEN
        _runOneStep := FALSE;
        RETURN;
    END_IF
END_IF

IF SUPER^.Step(202, TRUE, 'Step number 202') THEN
    SUPER^.StepCompleteWhen((_runOneStep OR _runAllSteps) AND _finishStep);

    IF _runOneStep THEN
        _runOneStep := FALSE;
        RETURN;
    END_IF
END_IF

IF SUPER^.Step(203, TRUE, 'Step number 203') THEN
    SUPER^.StepCompleteWhen((_runOneStep OR _runAllSteps) AND _finishStep);

    IF _runOneStep THEN
        _runOneStep := FALSE;
        RETURN;
    END_IF
END_IF

IF SUPER^.Step(204, TRUE, 'Step number 204') THEN
    SUPER^.StepCompleteWhen((_runOneStep OR _runAllSteps) AND _finishStep);

    IF _runOneStep THEN
        _runOneStep := FALSE;
        RETURN;
    END_IF
END_IF

IF SUPER^.Step(205, TRUE, 'Step number 205') THEN
    SUPER^.StepCompleteWhen((_runOneStep OR _runAllSteps) AND _finishStep);

    IF _runOneStep THEN
        _runOneStep := FALSE;
        RETURN;
    END_IF
END_IF

IF SUPER^.Step(206, TRUE, 'Step number 206') THEN
    SUPER^.StepCompleteWhen((_runOneStep OR _runAllSteps) AND _finishStep);

    IF _runOneStep THEN
        _runOneStep := FALSE;
        RETURN;
    END_IF
END_IF

IF SUPER^.Step(207, TRUE, 'Step number 207') THEN
    SUPER^.StepCompleteWhen((_runOneStep OR _runAllSteps) AND _finishStep);

    IF _runOneStep THEN
        _runOneStep := FALSE;
        RETURN;
    END_IF
END_IF

IF SUPER^.Step(208, TRUE, 'Step number 208') THEN
    SUPER^.StepCompleteWhen((_runOneStep OR _runAllSteps) AND _finishStep);

    IF _runOneStep THEN
        _runOneStep := FALSE;
        RETURN;
    END_IF
END_IF

IF SUPER^.Step(209, TRUE, 'Step number 209') THEN
    SUPER^.StepCompleteWhen((_runOneStep OR _runAllSteps) AND _finishStep);

    IF _runOneStep THEN
        _runOneStep := FALSE;
        RETURN;
    END_IF
END_IF

IF SUPER^.Step(210, TRUE, 'Step number 210') THEN
    SUPER^.StepCompleteWhen((_runOneStep OR _runAllSteps) AND _finishStep);

    IF _runOneStep THEN
        _runOneStep := FALSE;
        RETURN;
    END_IF
END_IF

IF SUPER^.Step(211, TRUE, 'Step number 211') THEN
    SUPER^.StepCompleteWhen((_runOneStep OR _runAllSteps) AND _finishStep);

    IF _runOneStep THEN
        _runOneStep := FALSE;
        RETURN;
    END_IF
END_IF

IF SUPER^.Step(212, TRUE, 'Step number 212') THEN
    SUPER^.StepCompleteWhen((_runOneStep OR _runAllSteps) AND _finishStep);

    IF _runOneStep THEN
        _runOneStep := FALSE;
        RETURN;
    END_IF
END_IF

IF SUPER^.Step(213, TRUE, 'Step number 213') THEN
    SUPER^.StepCompleteWhen((_runOneStep OR _runAllSteps) AND _finishStep);

    IF _runOneStep THEN
        _runOneStep := FALSE;
        RETURN;
    END_IF
END_IF

IF SUPER^.Step(214, TRUE, 'Step number 214') THEN
    SUPER^.StepCompleteWhen((_runOneStep OR _runAllSteps) AND _finishStep);

    IF _runOneStep THEN
        _runOneStep := FALSE;
        RETURN;
    END_IF
END_IF

IF SUPER^.Step(215, TRUE, 'Step number 215') THEN
    SUPER^.StepCompleteWhen((_runOneStep OR _runAllSteps) AND _finishStep);

    IF _runOneStep THEN
        _runOneStep := FALSE;
        RETURN;
    END_IF
END_IF

IF SUPER^.Step(216, TRUE, 'Step number 216') THEN
    SUPER^.StepCompleteWhen((_runOneStep OR _runAllSteps) AND _finishStep);

    IF _runOneStep THEN
        _runOneStep := FALSE;
        RETURN;
    END_IF
END_IF

IF SUPER^.Step(217, TRUE, 'Step number 217') THEN
    SUPER^.StepCompleteWhen((_runOneStep OR _runAllSteps) AND _finishStep);

    IF _runOneStep THEN
        _runOneStep := FALSE;
        RETURN;
    END_IF
END_IF

IF SUPER^.Step(218, TRUE, 'Step number 218') THEN
    SUPER^.StepCompleteWhen((_runOneStep OR _runAllSteps) AND _finishStep);

    IF _runOneStep THEN
        _runOneStep := FALSE;
        RETURN;
    END_IF
END_IF

IF SUPER^.Step(219, TRUE, 'Step number 219') THEN
    SUPER^.StepCompleteWhen((_runOneStep OR _runAllSteps) AND _finishStep);

    IF _runOneStep THEN
        _runOneStep := FALSE;
        RETURN;
    END_IF
END_IF

IF SUPER^.Step(220, TRUE, 'Step number 220') THEN
    SUPER^.StepCompleteWhen((_runOneStep OR _runAllSteps) AND _finishStep);

    IF _runOneStep THEN
        _runOneStep := FALSE;
        RETURN;
    END_IF
END_IF

IF SUPER^.Step(221, TRUE, 'Step number 221') THEN
    SUPER^.StepCompleteWhen((_runOneStep OR _runAllSteps) AND _finishStep);

    IF _runOneStep THEN
        _runOneStep := FALSE;
        RETURN;
    END_IF
END_IF

IF SUPER^.Step(222, TRUE, 'Step number 222') THEN
    SUPER^.StepCompleteWhen((_runOneStep OR _runAllSteps) AND _finishStep);

    IF _runOneStep THEN
        _runOneStep := FALSE;
        RETURN;
    END_IF
END_IF

IF SUPER^.Step(223, TRUE, 'Step number 223') THEN
    SUPER^.StepCompleteWhen((_runOneStep OR _runAllSteps) AND _finishStep);

    IF _runOneStep THEN
        _runOneStep := FALSE;
        RETURN;
    END_IF
END_IF

IF SUPER^.Step(224, TRUE, 'Step number 224') THEN
    SUPER^.StepCompleteWhen((_runOneStep OR _runAllSteps) AND _finishStep);

    IF _runOneStep THEN
        _runOneStep := FALSE;
        RETURN;
    END_IF
END_IF

IF SUPER^.Step(225, TRUE, 'Step number 225') THEN
    SUPER^.StepCompleteWhen((_runOneStep OR _runAllSteps) AND _finishStep);

    IF _runOneStep THEN
        _runOneStep := FALSE;
        RETURN;
    END_IF
END_IF

IF SUPER^.Step(226, TRUE, 'Step number 226') THEN
    SUPER^.StepCompleteWhen((_runOneStep OR _runAllSteps) AND _finishStep);

    IF _runOneStep THEN
        _runOneStep := FALSE;
        RETURN;
    END_IF
END_IF

IF SUPER^.Step(227, TRUE, 'Step number 227') THEN
    SUPER^.StepCompleteWhen((_runOneStep OR _runAllSteps) AND _finishStep);

    IF _runOneStep THEN
        _runOneStep := FALSE;
        RETURN;
    END_IF
END_IF

IF SUPER^.Step(228, TRUE, 'Step number 228') THEN
    SUPER^.StepCompleteWhen((_runOneStep OR _runAllSteps) AND _finishStep);

    IF _runOneStep THEN
        _runOneStep := FALSE;
        RETURN;
    END_IF
END_IF

IF SUPER^.Step(229, TRUE, 'Step number 229') THEN
    SUPER^.StepCompleteWhen((_runOneStep OR _runAllSteps) AND _finishStep);

    IF _runOneStep THEN
        _runOneStep := FALSE;
        RETURN;
    END_IF
END_IF

IF SUPER^.Step(230, TRUE, 'Step number 230') THEN
    SUPER^.StepCompleteWhen((_runOneStep OR _runAllSteps) AND _finishStep);

    IF _runOneStep THEN
        _runOneStep := FALSE;
        RETURN;
    END_IF
END_IF

IF SUPER^.Step(231, TRUE, 'Step number 231') THEN
    SUPER^.StepCompleteWhen((_runOneStep OR _runAllSteps) AND _finishStep);

    IF _runOneStep THEN
        _runOneStep := FALSE;
        RETURN;
    END_IF
END_IF

IF SUPER^.Step(232, TRUE, 'Step number 232') THEN
    SUPER^.StepCompleteWhen((_runOneStep OR _runAllSteps) AND _finishStep);

    IF _runOneStep THEN
        _runOneStep := FALSE;
        RETURN;
    END_IF
END_IF

IF SUPER^.Step(233, TRUE, 'Step number 233') THEN
    SUPER^.StepCompleteWhen((_runOneStep OR _runAllSteps) AND _finishStep);

    IF _runOneStep THEN
        _runOneStep := FALSE;
        RETURN;
    END_IF
END_IF

IF SUPER^.Step(234, TRUE, 'Step number 234') THEN
    SUPER^.StepCompleteWhen((_runOneStep OR _runAllSteps) AND _finishStep);

    IF _runOneStep THEN
        _runOneStep := FALSE;
        RETURN;
    END_IF
END_IF

IF SUPER^.Step(235, TRUE, 'Step number 235') THEN
    SUPER^.StepCompleteWhen((_runOneStep OR _runAllSteps) AND _finishStep);

    IF _runOneStep THEN
        _runOneStep := FALSE;
        RETURN;
    END_IF
END_IF

IF SUPER^.Step(236, TRUE, 'Step number 236') THEN
    SUPER^.StepCompleteWhen((_runOneStep OR _runAllSteps) AND _finishStep);

    IF _runOneStep THEN
        _runOneStep := FALSE;
        RETURN;
    END_IF
END_IF

IF SUPER^.Step(237, TRUE, 'Step number 237') THEN
    SUPER^.StepCompleteWhen((_runOneStep OR _runAllSteps) AND _finishStep);

    IF _runOneStep THEN
        _runOneStep := FALSE;
        RETURN;
    END_IF
END_IF

IF SUPER^.Step(238, TRUE, 'Step number 238') THEN
    SUPER^.StepCompleteWhen((_runOneStep OR _runAllSteps) AND _finishStep);

    IF _runOneStep THEN
        _runOneStep := FALSE;
        RETURN;
    END_IF
END_IF

IF SUPER^.Step(239, TRUE, 'Step number 239') THEN
    SUPER^.StepCompleteWhen((_runOneStep OR _runAllSteps) AND _finishStep);

    IF _runOneStep THEN
        _runOneStep := FALSE;
        RETURN;
    END_IF
END_IF

IF SUPER^.Step(240, TRUE, 'Step number 240') THEN
    SUPER^.StepCompleteWhen((_runOneStep OR _runAllSteps) AND _finishStep);

    IF _runOneStep THEN
        _runOneStep := FALSE;
        RETURN;
    END_IF
END_IF

IF SUPER^.Step(241, TRUE, 'Step number 241') THEN
    SUPER^.StepCompleteWhen((_runOneStep OR _runAllSteps) AND _finishStep);

    IF _runOneStep THEN
        _runOneStep := FALSE;
        RETURN;
    END_IF
END_IF

IF SUPER^.Step(242, TRUE, 'Step number 242') THEN
    SUPER^.StepCompleteWhen((_runOneStep OR _runAllSteps) AND _finishStep);

    IF _runOneStep THEN
        _runOneStep := FALSE;
        RETURN;
    END_IF
END_IF

IF SUPER^.Step(243, TRUE, 'Step number 243') THEN
    SUPER^.StepCompleteWhen((_runOneStep OR _runAllSteps) AND _finishStep);

    IF _runOneStep THEN
        _runOneStep := FALSE;
        RETURN;
    END_IF
END_IF

IF SUPER^.Step(244, TRUE, 'Step number 244') THEN
    SUPER^.StepCompleteWhen((_runOneStep OR _runAllSteps) AND _finishStep);

    IF _runOneStep THEN
        _runOneStep := FALSE;
        RETURN;
    END_IF
END_IF

IF SUPER^.Step(245, TRUE, 'Step number 245') THEN
    SUPER^.StepCompleteWhen((_runOneStep OR _runAllSteps) AND _finishStep);

    IF _runOneStep THEN
        _runOneStep := FALSE;
        RETURN;
    END_IF
END_IF

IF SUPER^.Step(246, TRUE, 'Step number 246') THEN
    SUPER^.StepCompleteWhen((_runOneStep OR _runAllSteps) AND _finishStep);

    IF _runOneStep THEN
        _runOneStep := FALSE;
        RETURN;
    END_IF
END_IF

IF SUPER^.Step(247, TRUE, 'Step number 247') THEN
    SUPER^.StepCompleteWhen((_runOneStep OR _runAllSteps) AND _finishStep);

    IF _runOneStep THEN
        _runOneStep := FALSE;
        RETURN;
    END_IF
END_IF

IF SUPER^.Step(248, TRUE, 'Step number 248') THEN
    SUPER^.StepCompleteWhen((_runOneStep OR _runAllSteps) AND _finishStep);

    IF _runOneStep THEN
        _runOneStep := FALSE;
        RETURN;
    END_IF
END_IF

IF SUPER^.Step(249, TRUE, 'Step number 249') THEN
    SUPER^.StepCompleteWhen((_runOneStep OR _runAllSteps) AND _finishStep);

    IF _runOneStep THEN
        _runOneStep := FALSE;
        RETURN;
    END_IF
END_IF

IF SUPER^.Step(250, TRUE, 'Step number 250') THEN
    SUPER^.StepCompleteWhen((_runOneStep OR _runAllSteps) AND _finishStep);

    IF _runOneStep THEN
        _runOneStep := FALSE;
        RETURN;
    END_IF
END_IF

IF SUPER^.Step(251, TRUE, 'Step number 251') THEN
    SUPER^.StepCompleteWhen((_runOneStep OR _runAllSteps) AND _finishStep);

    IF _runOneStep THEN
        _runOneStep := FALSE;
        RETURN;
    END_IF
END_IF

IF SUPER^.Step(252, TRUE, 'Step number 252') THEN
    SUPER^.StepCompleteWhen((_runOneStep OR _runAllSteps) AND _finishStep);

    IF _runOneStep THEN
        _runOneStep := FALSE;
        RETURN;
    END_IF
END_IF

IF SUPER^.Step(253, TRUE, 'Step number 253') THEN
    SUPER^.StepCompleteWhen((_runOneStep OR _runAllSteps) AND _finishStep);

    IF _runOneStep THEN
        _runOneStep := FALSE;
        RETURN;
    END_IF
END_IF

IF SUPER^.Step(254, TRUE, 'Step number 254') THEN
    SUPER^.StepCompleteWhen((_runOneStep OR _runAllSteps) AND _finishStep);

    IF _runOneStep THEN
        _runOneStep := FALSE;
        RETURN;
    END_IF
END_IF

IF SUPER^.Step(255, TRUE, 'Step number 255') THEN
    SUPER^.StepCompleteWhen((_runOneStep OR _runAllSteps) AND _finishStep);

    IF _runOneStep THEN
        _runOneStep := FALSE;
        RETURN;
    END_IF
END_IF

IF SUPER^.Step(256, TRUE, 'Step number 256') THEN
    SUPER^.StepCompleteWhen((_runOneStep OR _runAllSteps) AND _finishStep);

    IF _runOneStep THEN
        _runOneStep := FALSE;
        RETURN;
    END_IF
END_IF

IF SUPER^.Step(257, TRUE, 'Step number 257') THEN
    SUPER^.StepCompleteWhen((_runOneStep OR _runAllSteps) AND _finishStep);

    IF _runOneStep THEN
        _runOneStep := FALSE;
        RETURN;
    END_IF
END_IF

IF SUPER^.Step(258, TRUE, 'Step number 258') THEN
    SUPER^.StepCompleteWhen((_runOneStep OR _runAllSteps) AND _finishStep);

    IF _runOneStep THEN
        _runOneStep := FALSE;
        RETURN;
    END_IF
END_IF

IF SUPER^.Step(259, TRUE, 'Step number 259') THEN
    SUPER^.StepCompleteWhen((_runOneStep OR _runAllSteps) AND _finishStep);

    IF _runOneStep THEN
        _runOneStep := FALSE;
        RETURN;
    END_IF
END_IF

IF SUPER^.Step(260, TRUE, 'Step number 260') THEN
    SUPER^.StepCompleteWhen((_runOneStep OR _runAllSteps) AND _finishStep);

    IF _runOneStep THEN
        _runOneStep := FALSE;
        RETURN;
    END_IF
END_IF

IF SUPER^.Step(261, TRUE, 'Step number 261') THEN
    SUPER^.StepCompleteWhen((_runOneStep OR _runAllSteps) AND _finishStep);

    IF _runOneStep THEN
        _runOneStep := FALSE;
        RETURN;
    END_IF
END_IF

IF SUPER^.Step(262, TRUE, 'Step number 262') THEN
    SUPER^.StepCompleteWhen((_runOneStep OR _runAllSteps) AND _finishStep);

    IF _runOneStep THEN
        _runOneStep := FALSE;
        RETURN;
    END_IF
END_IF

IF SUPER^.Step(263, TRUE, 'Step number 263') THEN
    SUPER^.StepCompleteWhen((_runOneStep OR _runAllSteps) AND _finishStep);

    IF _runOneStep THEN
        _runOneStep := FALSE;
        RETURN;
    END_IF
END_IF

IF SUPER^.Step(264, TRUE, 'Step number 264') THEN
    SUPER^.StepCompleteWhen((_runOneStep OR _runAllSteps) AND _finishStep);

    IF _runOneStep THEN
        _runOneStep := FALSE;
        RETURN;
    END_IF
END_IF

IF SUPER^.Step(265, TRUE, 'Step number 265') THEN
    SUPER^.StepCompleteWhen((_runOneStep OR _runAllSteps) AND _finishStep);

    IF _runOneStep THEN
        _runOneStep := FALSE;
        RETURN;
    END_IF
END_IF

IF SUPER^.Step(266, TRUE, 'Step number 266') THEN
    SUPER^.StepCompleteWhen((_runOneStep OR _runAllSteps) AND _finishStep);

    IF _runOneStep THEN
        _runOneStep := FALSE;
        RETURN;
    END_IF
END_IF

IF SUPER^.Step(267, TRUE, 'Step number 267') THEN
    SUPER^.StepCompleteWhen((_runOneStep OR _runAllSteps) AND _finishStep);

    IF _runOneStep THEN
        _runOneStep := FALSE;
        RETURN;
    END_IF
END_IF

IF SUPER^.Step(268, TRUE, 'Step number 268') THEN
    SUPER^.StepCompleteWhen((_runOneStep OR _runAllSteps) AND _finishStep);

    IF _runOneStep THEN
        _runOneStep := FALSE;
        RETURN;
    END_IF
END_IF

IF SUPER^.Step(269, TRUE, 'Step number 269') THEN
    SUPER^.StepCompleteWhen((_runOneStep OR _runAllSteps) AND _finishStep);

    IF _runOneStep THEN
        _runOneStep := FALSE;
        RETURN;
    END_IF
END_IF

IF SUPER^.Step(270, TRUE, 'Step number 270') THEN
    SUPER^.StepCompleteWhen((_runOneStep OR _runAllSteps) AND _finishStep);

    IF _runOneStep THEN
        _runOneStep := FALSE;
        RETURN;
    END_IF
END_IF

IF SUPER^.Step(271, TRUE, 'Step number 271') THEN
    SUPER^.StepCompleteWhen((_runOneStep OR _runAllSteps) AND _finishStep);

    IF _runOneStep THEN
        _runOneStep := FALSE;
        RETURN;
    END_IF
END_IF

IF SUPER^.Step(272, TRUE, 'Step number 272') THEN
    SUPER^.StepCompleteWhen((_runOneStep OR _runAllSteps) AND _finishStep);

    IF _runOneStep THEN
        _runOneStep := FALSE;
        RETURN;
    END_IF
END_IF

IF SUPER^.Step(273, TRUE, 'Step number 273') THEN
    SUPER^.StepCompleteWhen((_runOneStep OR _runAllSteps) AND _finishStep);

    IF _runOneStep THEN
        _runOneStep := FALSE;
        RETURN;
    END_IF
END_IF

IF SUPER^.Step(274, TRUE, 'Step number 274') THEN
    SUPER^.StepCompleteWhen((_runOneStep OR _runAllSteps) AND _finishStep);

    IF _runOneStep THEN
        _runOneStep := FALSE;
        RETURN;
    END_IF
END_IF

IF SUPER^.Step(275, TRUE, 'Step number 275') THEN
    SUPER^.StepCompleteWhen((_runOneStep OR _runAllSteps) AND _finishStep);

    IF _runOneStep THEN
        _runOneStep := FALSE;
        RETURN;
    END_IF
END_IF

IF SUPER^.Step(276, TRUE, 'Step number 276') THEN
    SUPER^.StepCompleteWhen((_runOneStep OR _runAllSteps) AND _finishStep);

    IF _runOneStep THEN
        _runOneStep := FALSE;
        RETURN;
    END_IF
END_IF

IF SUPER^.Step(277, TRUE, 'Step number 277') THEN
    SUPER^.StepCompleteWhen((_runOneStep OR _runAllSteps) AND _finishStep);

    IF _runOneStep THEN
        _runOneStep := FALSE;
        RETURN;
    END_IF
END_IF

IF SUPER^.Step(278, TRUE, 'Step number 278') THEN
    SUPER^.StepCompleteWhen((_runOneStep OR _runAllSteps) AND _finishStep);

    IF _runOneStep THEN
        _runOneStep := FALSE;
        RETURN;
    END_IF
END_IF

IF SUPER^.Step(279, TRUE, 'Step number 279') THEN
    SUPER^.StepCompleteWhen((_runOneStep OR _runAllSteps) AND _finishStep);

    IF _runOneStep THEN
        _runOneStep := FALSE;
        RETURN;
    END_IF
END_IF

IF SUPER^.Step(280, TRUE, 'Step number 280') THEN
    SUPER^.StepCompleteWhen((_runOneStep OR _runAllSteps) AND _finishStep);

    IF _runOneStep THEN
        _runOneStep := FALSE;
        RETURN;
    END_IF
END_IF

IF SUPER^.Step(281, TRUE, 'Step number 281') THEN
    SUPER^.StepCompleteWhen((_runOneStep OR _runAllSteps) AND _finishStep);

    IF _runOneStep THEN
        _runOneStep := FALSE;
        RETURN;
    END_IF
END_IF

IF SUPER^.Step(282, TRUE, 'Step number 282') THEN
    SUPER^.StepCompleteWhen((_runOneStep OR _runAllSteps) AND _finishStep);

    IF _runOneStep THEN
        _runOneStep := FALSE;
        RETURN;
    END_IF
END_IF

IF SUPER^.Step(283, TRUE, 'Step number 283') THEN
    SUPER^.StepCompleteWhen((_runOneStep OR _runAllSteps) AND _finishStep);

